LIN {X 0,Y 446.497,Z 325.867,A -85,B 0,C 180,E1 -8839.301,E2 -8839.301} C_VEL
LIN {X 0,Y 446.419,Z 325.877,A -85,B 0,C 180,E1 -8842.199,E2 -8842.199} C_VEL
LIN {X 0,Y 446.45,Z 325.872,A -85,B 0,C 180,E1 -8845.152,E2 -8845.152} C_VEL
LIN {X 0,Y 446.485,Z 325.867,A -85,B 0,C 180,E1 -8848.178,E2 -8848.178} C_VEL
LIN {X 0,Y 446.418,Z 325.875,A -85,B 0,C 180,E1 -8851.774,E2 -8851.774} C_VEL
LIN {X 0,Y 446.422,Z 325.878,A -85,B 0,C 180,E1 -8854.523,E2 -8854.523} C_VEL
LIN {X 0,Y 446.412,Z 325.876,A -85,B 0,C 180,E1 -8858.078,E2 -8858.078} C_VEL
LIN {X 0,Y 446.425,Z 325.876,A -85,B 0,C 180,E1 -8860.917,E2 -8860.917} C_VEL
LIN {X 0,Y 446.398,Z 325.878,A -85,B 0,C 180,E1 -8863.846,E2 -8863.846} C_VEL
LIN {X 0,Y 446.397,Z 325.882,A -85,B 0,C 180,E1 -8866.403,E2 -8866.403} C_VEL
LIN {X 0,Y 446.425,Z 325.874,A -85,B 0,C 180,E1 -8869.082,E2 -8869.082} C_VEL
LIN {X 0,Y 446.429,Z 325.874,A -85,B 0,C 180,E1 -8871.918,E2 -8871.918} C_VEL
LIN {X 0,Y 446.428,Z 325.873,A -85,B 0,C 180,E1 -8875.477,E2 -8875.477} C_VEL
LIN {X 0,Y 446.414,Z 325.878,A -85,B 0,C 180,E1 -8878.699,E2 -8878.699} C_VEL
LIN {X 0,Y 446.482,Z 325.868,A -85,B 0,C 180,E1 -8881.821,E2 -8881.821} C_VEL
LIN {X 0,Y 446.455,Z 325.871,A -85,B 0,C 180,E1 -8884.848,E2 -8884.848} C_VEL
LIN {X 0,Y 446.445,Z 325.876,A -85,B 0,C 180,E1 -8888.245,E2 -8888.245} C_VEL
LIN {X 0,Y 446.455,Z 325.871,A -85,B 0,C 180,E1 -8891.649,E2 -8891.649} C_VEL
LIN {X 0,Y 446.505,Z 325.868,A -85,B 0,C 180,E1 -8894.48,E2 -8894.48} C_VEL
LIN {X 0,Y 446.466,Z 325.869,A -85,B 0,C 180,E1 -8895.187,E2 -8895.187} C_VEL
LIN {X 0,Y 445.802,Z 325.955,A -85,B 0,C 180,E1 -8895.94,E2 -8895.94} C_VEL
LIN {X 0,Y 442.952,Z 326.308,A -85,B 0,C 180,E1 -8897.164,E2 -8897.164} C_VEL
LIN {X 0,Y 440.542,Z 326.611,A -85,B 0,C 180,E1 -8898.152,E2 -8898.152} C_VEL
LIN {X 0,Y 439.512,Z 326.735,A -85,B 0,C 180,E1 -8898.915,E2 -8898.915} C_VEL
LIN {X 0,Y 439.43,Z 326.745,A -85,B 0,C 180,E1 -8899.173,E2 -8899.173} C_VEL
LIN {X 0,Y 439.599,Z 326.726,A -85,B 0,C 180,E1 -8902.652,E2 -8902.652} C_VEL
LIN {X 0,Y 439.618,Z 326.725,A -85,B 0,C 180,E1 -8904.496,E2 -8904.496} C_VEL
LIN {X 0,Y 439.633,Z 326.725,A -85,B 0,C 180,E1 -8908.168,E2 -8908.168} C_VEL
LIN {X 0,Y 439.762,Z 326.708,A -85,B 0,C 180,E1 -8910,E2 -8910} C_VEL
LIN {X 0,Y 439.653,Z 326.718,A -85,B 0,C 180,E1 -8912.749,E2 -8912.749} C_VEL
LIN {X 0,Y 439.616,Z 326.725,A -85,B 0,C 180,E1 -8916.425,E2 -8916.425} C_VEL
LIN {X 0,Y 439.497,Z 326.738,A -85,B 0,C 180,E1 -8919.202,E2 -8919.202} C_VEL
LIN {X 0,Y 439.463,Z 326.741,A -85,B 0,C 180,E1 -8922.938,E2 -8922.938} C_VEL
LIN {X 0,Y 439.445,Z 326.746,A -85,B 0,C 180,E1 -8926.349,E2 -8926.349} C_VEL
LIN {X 0,Y 439.401,Z 326.751,A -85,B 0,C 180,E1 -8929.627,E2 -8929.627} C_VEL
LIN {X 0,Y 439.364,Z 326.754,A -85,B 0,C 180,E1 -8932.576,E2 -8932.576} C_VEL
LIN {X 0,Y 439.404,Z 326.751,A -85,B 0,C 180,E1 -8935.585,E2 -8935.585} C_VEL
LIN {X 0,Y 439.416,Z 326.747,A -85,B 0,C 180,E1 -8938.674,E2 -8938.674} C_VEL
LIN {X 0,Y 439.369,Z 326.757,A -85,B 0,C 180,E1 -8942.031,E2 -8942.031} C_VEL
LIN {X 0,Y 439.395,Z 326.751,A -85,B 0,C 180,E1 -8945.341,E2 -8945.341} C_VEL
LIN {X 0,Y 439.39,Z 326.751,A -85,B 0,C 180,E1 -8948.595,E2 -8948.595} C_VEL
LIN {X 0,Y 439.388,Z 326.752,A -85,B 0,C 180,E1 -8951.257,E2 -8951.257} C_VEL
LIN {X 0,Y 439.4,Z 326.75,A -85,B 0,C 180,E1 -8954.73,E2 -8954.73} C_VEL
LIN {X 0,Y 439.396,Z 326.755,A -85,B 0,C 180,E1 -8957.796,E2 -8957.796} C_VEL
LIN {X 0,Y 439.395,Z 326.751,A -85,B 0,C 180,E1 -8960.225,E2 -8960.225} C_VEL
LIN {X 0,Y 439.374,Z 326.758,A -85,B 0,C 180,E1 -8963.713,E2 -8963.713} C_VEL
LIN {X 0,Y 439.373,Z 326.754,A -85,B 0,C 180,E1 -8967.055,E2 -8967.055} C_VEL
LIN {X 0,Y 439.384,Z 326.752,A -85,B 0,C 180,E1 -8970.275,E2 -8970.275} C_VEL
LIN {X 0,Y 439.431,Z 326.749,A -85,B 0,C 180,E1 -8973.397,E2 -8973.397} C_VEL
LIN {X 0,Y 439.443,Z 326.743,A -85,B 0,C 180,E1 -8974.537,E2 -8974.537} C_VEL
LIN {X 0,Y 443.588,Z 339.182,A -85,B 0,C 180,E1 -8974.94,E2 -8974.94} C_VEL
LIN {X 0,Y 442.677,Z 414.373,A -85,B 0,C 180,E1 -8976.337,E2 -8976.337} C_VEL
LIN {X 0,Y 442.558,Z 425.989,A -85,B 0,C 180,E1 -8976.705,E2 -8976.705} C_VEL
LIN {X 0,Y 442.258,Z 438.78,A -85,B 0,C 180,E1 -8977.289,E2 -8977.289} C_VEL
LIN {X 0,Y 441.891,Z 451.182,A -85,B 0,C 180,E1 -8978.053,E2 -8978.053} C_VEL
LIN {X 0,Y 441.469,Z 461.829,A -85,B 0,C 180,E1 -8978.889,E2 -8978.889} C_VEL
LIN {X 0,Y 441.016,Z 472.96,A -85,B 0,C 180,E1 -8979.992,E2 -8979.992} C_VEL
LIN {X 0,Y 440.528,Z 482.488,A -85,B 0,C 180,E1 -8981.152,E2 -8981.152} C_VEL
LIN {X 0,Y 440.14,Z 490.434,A -85,B 0,C 180,E1 -8982.339,E2 -8982.339} C_VEL
LIN {X 0,Y 439.742,Z 498.632,A -85,B 0,C 180,E1 -8983.864,E2 -8983.864} C_VEL
LIN {X 0,Y 439.467,Z 504.268,A -85,B 0,C 180,E1 -8985.175,E2 -8985.175} C_VEL
LIN {X 0,Y 439.241,Z 509.068,A -85,B 0,C 180,E1 -8986.585,E2 -8986.585} C_VEL
LIN {X 0,Y 439.14,Z 512.67,A -85,B 0,C 180,E1 -8987.992,E2 -8987.992} C_VEL
LIN {X 0,Y 438.993,Z 514.461,A -85,B 0,C 180,E1 -8988.924,E2 -8988.924} C_VEL
LIN {X 0,Y 438.964,Z 515.833,A -85,B 0,C 180,E1 -8989.857,E2 -8989.857} C_VEL
LIN {X 0,Y 438.965,Z 516.774,A -85,B 0,C 180,E1 -8990.788,E2 -8990.788} C_VEL
LIN {X 0,Y 438.98,Z 517.257,A -85,B 0,C 180,E1 -8991.716,E2 -8991.716} C_VEL
LIN {X 0,Y 439.074,Z 517.293,A -85,B 0,C 180,E1 -8992.935,E2 -8992.935} C_VEL
LIN {X 0,Y 439.118,Z 516.257,A -85,B 0,C 180,E1 -8994.49,E2 -8994.49} C_VEL
LIN {X 0,Y 439.143,Z 515.092,A -85,B 0,C 180,E1 -8995.411,E2 -8995.411} C_VEL
LIN {X 0,Y 439.278,Z 512.524,A -85,B 0,C 180,E1 -8996.79,E2 -8996.79} C_VEL
LIN {X 0,Y 439.584,Z 508.903,A -85,B 0,C 180,E1 -8998.168,E2 -8998.168} C_VEL
LIN {X 0,Y 439.885,Z 504.163,A -85,B 0,C 180,E1 -8999.543,E2 -8999.543} C_VEL
LIN {X 0,Y 440.318,Z 498.125,A -85,B 0,C 180,E1 -9000.915,E2 -9000.915} C_VEL
LIN {X 0,Y 440.757,Z 490.589,A -85,B 0,C 180,E1 -9002.285,E2 -9002.285} C_VEL
LIN {X 0,Y 441.354,Z 481.185,A -85,B 0,C 180,E1 -9003.652,E2 -9003.652} C_VEL
LIN {X 0,Y 441.879,Z 471.347,A -85,B 0,C 180,E1 -9004.79,E2 -9004.79} C_VEL
LIN {X 0,Y 442.315,Z 460.406,A -85,B 0,C 180,E1 -9005.814,E2 -9005.814} C_VEL
LIN {X 0,Y 442.823,Z 449.541,A -85,B 0,C 180,E1 -9006.608,E2 -9006.608} C_VEL
LIN {X 0,Y 443.165,Z 436.449,A -85,B 0,C 180,E1 -9007.346,E2 -9007.346} C_VEL
LIN {X 0,Y 443.35,Z 423.637,A -85,B 0,C 180,E1 -9007.859,E2 -9007.859} C_VEL
LIN {X 0,Y 443.436,Z 410.181,A -85,B 0,C 180,E1 -9008.201,E2 -9008.201} C_VEL
LIN {X 0,Y 444.635,Z 339.873,A -85,B 0,C 180,E1 -9009.574,E2 -9009.574} C_VEL
LIN {X 0,Y 439.557,Z 327.4,A -85,B 0,C 180,E1 -9010.117,E2 -9010.117} C_VEL
LIN {X 0,Y 439.434,Z 326.752,A -85,B 0,C 180,E1 -9010.162,E2 -9010.162} C_VEL
LIN {X 0,Y 439.469,Z 326.745,A -85,B 0,C 180,E1 -9012.938,E2 -9012.938} C_VEL
LIN {X 0,Y 439.448,Z 326.747,A -85,B 0,C 180,E1 -9016.347,E2 -9016.347} C_VEL
LIN {X 0,Y 439.373,Z 326.757,A -85,B 0,C 180,E1 -9019.628,E2 -9019.628} C_VEL
LIN {X 0,Y 439.356,Z 326.757,A -85,B 0,C 180,E1 -9022.576,E2 -9022.576} C_VEL
LIN {X 0,Y 439.357,Z 326.757,A -85,B 0,C 180,E1 -9025.588,E2 -9025.588} C_VEL
LIN {X 0,Y 439.385,Z 326.753,A -85,B 0,C 180,E1 -9028.676,E2 -9028.676} C_VEL
LIN {X 0,Y 439.367,Z 326.757,A -85,B 0,C 180,E1 -9032.029,E2 -9032.029} C_VEL
LIN {X 0,Y 439.39,Z 326.748,A -85,B 0,C 180,E1 -9035.339,E2 -9035.339} C_VEL
LIN {X 0,Y 439.358,Z 326.753,A -85,B 0,C 180,E1 -9038.598,E2 -9038.598} C_VEL
LIN {X 0,Y 439.352,Z 326.756,A -85,B 0,C 180,E1 -9042.21,E2 -9042.21} C_VEL
LIN {X 0,Y 439.38,Z 326.753,A -85,B 0,C 180,E1 -9045.267,E2 -9045.267} C_VEL
LIN {X 0,Y 439.371,Z 326.752,A -85,B 0,C 180,E1 -9048.746,E2 -9048.746} C_VEL
LIN {X 0,Y 439.367,Z 326.758,A -85,B 0,C 180,E1 -9051.61,E2 -9051.61} C_VEL
LIN {X 0,Y 439.399,Z 326.75,A -85,B 0,C 180,E1 -9054.844,E2 -9054.844} C_VEL
LIN {X 0,Y 439.376,Z 326.754,A -85,B 0,C 180,E1 -9058.139,E2 -9058.139} C_VEL
LIN {X 0,Y 439.421,Z 326.85,A -85,B 0,C 180,E1 -9059.249,E2 -9059.249} C_VEL
LIN {X 0,Y 443.204,Z 343.947,A -85,B 0,C 180,E1 -9062.109,E2 -9062.109} C_VEL
LIN {X 0,Y 443.563,Z 347.321,A -85,B 0,C 180,E1 -9062.646,E2 -9062.646} C_VEL
LIN {X 0,Y 442.316,Z 368.721,A -85,B 0,C 180,E1 -9065.849,E2 -9065.849} C_VEL
LIN {X 0,Y 441.289,Z 388.385,A -85,B 0,C 180,E1 -9068.757,E2 -9068.757} C_VEL
LIN {X 0,Y 440.388,Z 409.595,A -85,B 0,C 180,E1 -9071.869,E2 -9071.869} C_VEL
LIN {X 0,Y 440.361,Z 410.41,A -85,B 0,C 180,E1 -9071.988,E2 -9071.988} C_VEL
LIN {X 0,Y 443.42,Z 438.789,A -85,B 0,C 180,E1 -9072.667,E2 -9072.667} C_VEL
LIN {X 0,Y 442.262,Z 521.633,A -85,B 0,C 180,E1 -9074.238,E2 -9074.238} C_VEL
LIN {X 0,Y 441.733,Z 534.688,A -85,B 0,C 180,E1 -9074.662,E2 -9074.662} C_VEL
LIN {X 0,Y 441.242,Z 546.877,A -85,B 0,C 180,E1 -9075.235,E2 -9075.235} C_VEL
LIN {X 0,Y 440.562,Z 559.508,A -85,B 0,C 180,E1 -9076.038,E2 -9076.038} C_VEL
LIN {X 0,Y 439.985,Z 571.311,A -85,B 0,C 180,E1 -9077.001,E2 -9077.001} C_VEL
LIN {X 0,Y 439.692,Z 580.107,A -85,B 0,C 180,E1 -9077.89,E2 -9077.89} C_VEL
LIN {X 0,Y 439.273,Z 588.726,A -85,B 0,C 180,E1 -9078.931,E2 -9078.931} C_VEL
LIN {X 0,Y 438.883,Z 598.064,A -85,B 0,C 180,E1 -9080.32,E2 -9080.32} C_VEL
LIN {X 0,Y 438.701,Z 605.586,A -85,B 0,C 180,E1 -9081.71,E2 -9081.71} C_VEL
LIN {X 0,Y 438.643,Z 611.595,A -85,B 0,C 180,E1 -9083.099,E2 -9083.099} C_VEL
LIN {X 0,Y 438.6,Z 616.273,A -85,B 0,C 180,E1 -9084.483,E2 -9084.483} C_VEL
LIN {X 0,Y 438.706,Z 618.729,A -85,B 0,C 180,E1 -9085.406,E2 -9085.406} C_VEL
LIN {X 0,Y 438.79,Z 620.721,A -85,B 0,C 180,E1 -9086.327,E2 -9086.327} C_VEL
LIN {X 0,Y 438.681,Z 622.237,A -85,B 0,C 180,E1 -9087.245,E2 -9087.245} C_VEL
LIN {X 0,Y 438.655,Z 623.274,A -85,B 0,C 180,E1 -9088.164,E2 -9088.164} C_VEL
LIN {X 0,Y 438.669,Z 623.889,A -85,B 0,C 180,E1 -9089.082,E2 -9089.082} C_VEL
LIN {X 0,Y 438.698,Z 624.084,A -85,B 0,C 180,E1 -9090,E2 -9090} C_VEL
LIN {X 0,Y 438.675,Z 623.83,A -85,B 0,C 180,E1 -9090.918,E2 -9090.918} C_VEL
LIN {X 0,Y 438.67,Z 623.115,A -85,B 0,C 180,E1 -9091.836,E2 -9091.836} C_VEL
LIN {X 0,Y 438.699,Z 621.982,A -85,B 0,C 180,E1 -9092.755,E2 -9092.755} C_VEL
LIN {X 0,Y 438.747,Z 619.435,A -85,B 0,C 180,E1 -9094.133,E2 -9094.133} C_VEL
LIN {X 0,Y 438.653,Z 615.806,A -85,B 0,C 180,E1 -9095.516,E2 -9095.516} C_VEL
LIN {X 0,Y 438.676,Z 610.23,A -85,B 0,C 180,E1 -9097.109,E2 -9097.109} C_VEL
LIN {X 0,Y 438.775,Z 603.838,A -85,B 0,C 180,E1 -9098.52,E2 -9098.52} C_VEL
LIN {X 0,Y 438.915,Z 595.986,A -85,B 0,C 180,E1 -9099.912,E2 -9099.912} C_VEL
LIN {X 0,Y 439.305,Z 586.319,A -85,B 0,C 180,E1 -9101.302,E2 -9101.302} C_VEL
LIN {X 0,Y 439.832,Z 576.403,A -85,B 0,C 180,E1 -9102.45,E2 -9102.45} C_VEL
LIN {X 0,Y 440.242,Z 567.168,A -85,B 0,C 180,E1 -9103.337,E2 -9103.337} C_VEL
LIN {X 0,Y 440.754,Z 556.383,A -85,B 0,C 180,E1 -9104.191,E2 -9104.191} C_VEL
LIN {X 0,Y 441.517,Z 543.551,A -85,B 0,C 180,E1 -9104.991,E2 -9104.991} C_VEL
LIN {X 0,Y 442.098,Z 530.571,A -85,B 0,C 180,E1 -9105.59,E2 -9105.59} C_VEL
LIN {X 0,Y 442.691,Z 516.243,A -85,B 0,C 180,E1 -9106.042,E2 -9106.042} C_VEL
LIN {X 0,Y 443.861,Z 437.805,A -85,B 0,C 180,E1 -9107.594,E2 -9107.594} C_VEL
LIN {X 0,Y 441.293,Z 411.851,A -85,B 0,C 180,E1 -9108.282,E2 -9108.282} C_VEL
LIN {X 0,Y 440.287,Z 404.18,A -85,B 0,C 180,E1 -9108.518,E2 -9108.518} C_VEL
LIN {X 0,Y 441.456,Z 379.504,A -85,B 0,C 180,E1 -9112.216,E2 -9112.216} C_VEL
LIN {X 0,Y 442.689,Z 357.498,A -85,B 0,C 180,E1 -9115.633,E2 -9115.633} C_VEL
LIN {X 0,Y 443.47,Z 345.209,A -85,B 0,C 180,E1 -9117.616,E2 -9117.616} C_VEL
LIN {X 0,Y 441.409,Z 334.678,A -85,B 0,C 180,E1 -9119.576,E2 -9119.576} C_VEL
LIN {X 0,Y 439.406,Z 326.756,A -85,B 0,C 180,E1 -9121.186,E2 -9121.186} C_VEL
LIN {X 0,Y 439.387,Z 326.756,A -85,B 0,C 180,E1 -9124.044,E2 -9124.044} C_VEL
LIN {X 0,Y 439.349,Z 326.759,A -85,B 0,C 180,E1 -9126.886,E2 -9126.886} C_VEL
LIN {X 0,Y 439.35,Z 326.76,A -85,B 0,C 180,E1 -9129.84,E2 -9129.84} C_VEL
LIN {X 0,Y 439.345,Z 326.76,A -85,B 0,C 180,E1 -9132.621,E2 -9132.621} C_VEL
LIN {X 0,Y 439.4,Z 326.751,A -85,B 0,C 180,E1 -9135.27,E2 -9135.27} C_VEL
LIN {X 0,Y 439.358,Z 326.755,A -85,B 0,C 180,E1 -9139.016,E2 -9139.016} C_VEL
LIN {X 0,Y 439.337,Z 326.757,A -85,B 0,C 180,E1 -9142.563,E2 -9142.563} C_VEL
LIN {X 0,Y 439.393,Z 326.75,A -85,B 0,C 180,E1 -9144.843,E2 -9144.843} C_VEL
LIN {X 0,Y 439.368,Z 326.757,A -85,B 0,C 180,E1 -9148.139,E2 -9148.139} C_VEL
LIN {X 0,Y 439.388,Z 326.755,A -85,B 0,C 180,E1 -9151.609,E2 -9151.609} C_VEL
LIN {X 0,Y 439.355,Z 326.758,A -85,B 0,C 180,E1 -9154.412,E2 -9154.412} C_VEL
LIN {X 0,Y 439.355,Z 326.761,A -85,B 0,C 180,E1 -9157.424,E2 -9157.424} C_VEL
LIN {X 0,Y 439.388,Z 326.754,A -85,B 0,C 180,E1 -9160.684,E2 -9160.684} C_VEL
LIN {X 0,Y 439.473,Z 326.747,A -85,B 0,C 180,E1 -9163.835,E2 -9163.835} C_VEL
LIN {X 0,Y 440.548,Z 329.721,A -85,B 0,C 180,E1 -9163.975,E2 -9163.975} C_VEL
LIN {X 0,Y 444.907,Z 340.719,A -85,B 0,C 180,E1 -9164.47,E2 -9164.47} C_VEL
LIN {X 0,Y 443.421,Z 417.623,A -85,B 0,C 180,E1 -9166.042,E2 -9166.042} C_VEL
LIN {X 0,Y 443.277,Z 431.324,A -85,B 0,C 180,E1 -9166.505,E2 -9166.505} C_VEL
LIN {X 0,Y 443.021,Z 443.747,A -85,B 0,C 180,E1 -9167.109,E2 -9167.109} C_VEL
LIN {X 0,Y 442.706,Z 455.181,A -85,B 0,C 180,E1 -9167.857,E2 -9167.857} C_VEL
LIN {X 0,Y 442.146,Z 466.263,A -85,B 0,C 180,E1 -9168.771,E2 -9168.771} C_VEL
LIN {X 0,Y 441.664,Z 476.26,A -85,B 0,C 180,E1 -9169.803,E2 -9169.803} C_VEL
LIN {X 0,Y 441.182,Z 484.458,A -85,B 0,C 180,E1 -9170.833,E2 -9170.833} C_VEL
LIN {X 0,Y 440.621,Z 493.308,A -85,B 0,C 180,E1 -9172.208,E2 -9172.208} C_VEL
LIN {X 0,Y 440.208,Z 500.393,A -85,B 0,C 180,E1 -9173.583,E2 -9173.583} C_VEL
LIN {X 0,Y 439.806,Z 506.032,A -85,B 0,C 180,E1 -9174.957,E2 -9174.957} C_VEL
LIN {X 0,Y 439.444,Z 510.432,A -85,B 0,C 180,E1 -9176.332,E2 -9176.332} C_VEL
LIN {X 0,Y 439.271,Z 512.716,A -85,B 0,C 180,E1 -9177.248,E2 -9177.248} C_VEL
LIN {X 0,Y 439.295,Z 514.538,A -85,B 0,C 180,E1 -9178.166,E2 -9178.166} C_VEL
LIN {X 0,Y 439.151,Z 515.963,A -85,B 0,C 180,E1 -9179.083,E2 -9179.083} C_VEL
LIN {X 0,Y 439.083,Z 516.914,A -85,B 0,C 180,E1 -9180,E2 -9180} C_VEL
LIN {X 0,Y 439.069,Z 517.457,A -85,B 0,C 180,E1 -9180.917,E2 -9180.917} C_VEL
LIN {X 0,Y 438.841,Z 517.636,A -85,B 0,C 180,E1 -9181.835,E2 -9181.835} C_VEL
LIN {X 0,Y 438.868,Z 517.357,A -85,B 0,C 180,E1 -9182.753,E2 -9182.753} C_VEL
LIN {X 0,Y 439.079,Z 515.522,A -85,B 0,C 180,E1 -9184.59,E2 -9184.59} C_VEL
LIN {X 0,Y 439.171,Z 513.052,A -85,B 0,C 180,E1 -9185.97,E2 -9185.97} C_VEL
LIN {X 0,Y 439.307,Z 509.56,A -85,B 0,C 180,E1 -9187.353,E2 -9187.353} C_VEL
LIN {X 0,Y 439.482,Z 504.951,A -85,B 0,C 180,E1 -9188.738,E2 -9188.738} C_VEL
LIN {X 0,Y 439.724,Z 499.09,A -85,B 0,C 180,E1 -9190.125,E2 -9190.125} C_VEL
LIN {X 0,Y 440.091,Z 491.706,A -85,B 0,C 180,E1 -9191.514,E2 -9191.514} C_VEL
LIN {X 0,Y 440.535,Z 482.494,A -85,B 0,C 180,E1 -9192.905,E2 -9192.905} C_VEL
LIN {X 0,Y 440.919,Z 472.98,A -85,B 0,C 180,E1 -9194.068,E2 -9194.068} C_VEL
LIN {X 0,Y 441.452,Z 462.355,A -85,B 0,C 180,E1 -9195.111,E2 -9195.111} C_VEL
LIN {X 0,Y 441.831,Z 450.551,A -85,B 0,C 180,E1 -9196.044,E2 -9196.044} C_VEL
LIN {X 0,Y 442.304,Z 438.038,A -85,B 0,C 180,E1 -9196.797,E2 -9196.797} C_VEL
LIN {X 0,Y 442.521,Z 424.952,A -85,B 0,C 180,E1 -9197.384,E2 -9197.384} C_VEL
LIN {X 0,Y 442.633,Z 412.315,A -85,B 0,C 180,E1 -9197.766,E2 -9197.766} C_VEL
LIN {X 0,Y 443.576,Z 339.103,A -85,B 0,C 180,E1 -9199.137,E2 -9199.137} C_VEL
LIN {X 0,Y 439.436,Z 326.746,A -85,B 0,C 180,E1 -9199.535,E2 -9199.535} C_VEL
LIN {X 0,Y 439.366,Z 326.758,A -85,B 0,C 180,E1 -9202.575,E2 -9202.575} C_VEL
LIN {X 0,Y 439.401,Z 326.748,A -85,B 0,C 180,E1 -9205.585,E2 -9205.585} C_VEL
LIN {X 0,Y 439.417,Z 326.752,A -85,B 0,C 180,E1 -9208.673,E2 -9208.673} C_VEL
LIN {X 0,Y 439.368,Z 326.753,A -85,B 0,C 180,E1 -9212.03,E2 -9212.03} C_VEL
LIN {X 0,Y 439.391,Z 326.75,A -85,B 0,C 180,E1 -9215.339,E2 -9215.339} C_VEL
LIN {X 0,Y 439.374,Z 326.758,A -85,B 0,C 180,E1 -9218.595,E2 -9218.595} C_VEL
LIN {X 0,Y 439.387,Z 326.751,A -85,B 0,C 180,E1 -9221.256,E2 -9221.256} C_VEL
LIN {X 0,Y 439.398,Z 326.753,A -85,B 0,C 180,E1 -9224.729,E2 -9224.729} C_VEL
LIN {X 0,Y 439.394,Z 326.75,A -85,B 0,C 180,E1 -9227.795,E2 -9227.795} C_VEL
LIN {X 0,Y 439.435,Z 326.747,A -85,B 0,C 180,E1 -9230.228,E2 -9230.228} C_VEL
LIN {X 0,Y 439.375,Z 326.752,A -85,B 0,C 180,E1 -9233.713,E2 -9233.713} C_VEL
LIN {X 0,Y 439.37,Z 326.753,A -85,B 0,C 180,E1 -9237.054,E2 -9237.054} C_VEL
LIN {X 0,Y 439.38,Z 326.755,A -85,B 0,C 180,E1 -9240.274,E2 -9240.274} C_VEL
LIN {X 0,Y 439.427,Z 326.746,A -85,B 0,C 180,E1 -9243.396,E2 -9243.396} C_VEL
LIN {X 0,Y 439.385,Z 326.756,A -85,B 0,C 180,E1 -9246.43,E2 -9246.43} C_VEL
LIN {X 0,Y 439.386,Z 326.751,A -85,B 0,C 180,E1 -9249.397,E2 -9249.397} C_VEL
LIN {X 0,Y 439.429,Z 326.751,A -85,B 0,C 180,E1 -9252.309,E2 -9252.309} C_VEL
LIN {X 0,Y 439.445,Z 326.743,A -85,B 0,C 180,E1 -9255.176,E2 -9255.176} C_VEL
LIN {X 0,Y 439.481,Z 326.742,A -85,B 0,C 180,E1 -9258.001,E2 -9258.001} C_VEL
LIN {X 0,Y 439.43,Z 326.745,A -85,B 0,C 180,E1 -9259.173,E2 -9259.173} C_VEL
LIN {X 0,Y 438.78,Z 326.83,A -85,B 0,C 180,E1 -9259.939,E2 -9259.939} C_VEL
LIN {X 0,Y 435.978,Z 327.175,A -85,B 0,C 180,E1 -9261.184,E2 -9261.184} C_VEL
LIN {X 0,Y 433.619,Z 327.474,A -85,B 0,C 180,E1 -9262.189,E2 -9262.189} C_VEL
LIN {X 0,Y 432.627,Z 327.593,A -85,B 0,C 180,E1 -9262.965,E2 -9262.965} C_VEL
LIN {X 0,Y 432.557,Z 327.601,A -85,B 0,C 180,E1 -9263.227,E2 -9263.227} C_VEL
LIN {X 0,Y 432.398,Z 327.622,A -85,B 0,C 180,E1 -9265.339,E2 -9265.339} C_VEL
LIN {X 0,Y 432.603,Z 327.6,A -85,B 0,C 180,E1 -9268.138,E2 -9268.138} C_VEL
LIN {X 0,Y 432.731,Z 327.583,A -85,B 0,C 180,E1 -9270,E2 -9270} C_VEL
LIN {X 0,Y 432.602,Z 327.596,A -85,B 0,C 180,E1 -9272.794,E2 -9272.794} C_VEL
LIN {X 0,Y 432.57,Z 327.602,A -85,B 0,C 180,E1 -9276.531,E2 -9276.531} C_VEL
LIN {X 0,Y 432.44,Z 327.617,A -85,B 0,C 180,E1 -9279.353,E2 -9279.353} C_VEL
LIN {X 0,Y 432.428,Z 327.618,A -85,B 0,C 180,E1 -9282.804,E2 -9282.804} C_VEL
LIN {X 0,Y 432.41,Z 327.621,A -85,B 0,C 180,E1 -9286.479,E2 -9286.479} C_VEL
LIN {X 0,Y 432.337,Z 327.634,A -85,B 0,C 180,E1 -9289.961,E2 -9289.961} C_VEL
LIN {X 0,Y 432.318,Z 327.632,A -85,B 0,C 180,E1 -9292.965,E2 -9292.965} C_VEL
LIN {X 0,Y 432.363,Z 327.63,A -85,B 0,C 180,E1 -9296.033,E2 -9296.033} C_VEL
LIN {X 0,Y 432.342,Z 327.629,A -85,B 0,C 180,E1 -9299.188,E2 -9299.188} C_VEL
LIN {X 0,Y 432.322,Z 327.632,A -85,B 0,C 180,E1 -9302.443,E2 -9302.443} C_VEL
LIN {X 0,Y 432.345,Z 327.631,A -85,B 0,C 180,E1 -9305.633,E2 -9305.633} C_VEL
LIN {X 0,Y 432.352,Z 327.628,A -85,B 0,C 180,E1 -9308.717,E2 -9308.717} C_VEL
LIN {X 0,Y 432.334,Z 327.634,A -85,B 0,C 180,E1 -9311.798,E2 -9311.798} C_VEL
LIN {X 0,Y 432.333,Z 327.63,A -85,B 0,C 180,E1 -9314.348,E2 -9314.348} C_VEL
LIN {X 0,Y 432.32,Z 327.632,A -85,B 0,C 180,E1 -9317.016,E2 -9317.016} C_VEL
LIN {X 0,Y 432.334,Z 327.634,A -85,B 0,C 180,E1 -9319.821,E2 -9319.821} C_VEL
LIN {X 0,Y 432.307,Z 327.634,A -85,B 0,C 180,E1 -9323.023,E2 -9323.023} C_VEL
LIN {X 0,Y 432.359,Z 327.629,A -85,B 0,C 180,E1 -9325.998,E2 -9325.998} C_VEL
LIN {X 0,Y 432.349,Z 327.631,A -85,B 0,C 180,E1 -9329.49,E2 -9329.49} C_VEL
LIN {X 0,Y 432.393,Z 327.624,A -85,B 0,C 180,E1 -9332.929,E2 -9332.929} C_VEL
LIN {X 0,Y 432.45,Z 327.759,A -85,B 0,C 180,E1 -9334.315,E2 -9334.315} C_VEL
LIN {X 0,Y 436.747,Z 340.599,A -85,B 0,C 180,E1 -9334.725,E2 -9334.725} C_VEL
LIN {X 0,Y 435.769,Z 414.594,A -85,B 0,C 180,E1 -9336.128,E2 -9336.128} C_VEL
LIN {X 0,Y 435.651,Z 425.89,A -85,B 0,C 180,E1 -9336.484,E2 -9336.484} C_VEL
LIN {X 0,Y 435.375,Z 438.76,A -85,B 0,C 180,E1 -9337.066,E2 -9337.066} C_VEL
LIN {X 0,Y 434.987,Z 450.886,A -85,B 0,C 180,E1 -9337.811,E2 -9337.811} C_VEL
LIN {X 0,Y 434.548,Z 461.754,A -85,B 0,C 180,E1 -9338.661,E2 -9338.661} C_VEL
LIN {X 0,Y 434.129,Z 471.956,A -85,B 0,C 180,E1 -9339.654,E2 -9339.654} C_VEL
LIN {X 0,Y 433.612,Z 481.837,A -85,B 0,C 180,E1 -9340.84,E2 -9340.84} C_VEL
LIN {X 0,Y 433.179,Z 490.076,A -85,B 0,C 180,E1 -9342.046,E2 -9342.046} C_VEL
LIN {X 0,Y 432.817,Z 497.339,A -85,B 0,C 180,E1 -9343.343,E2 -9343.343} C_VEL
LIN {X 0,Y 432.465,Z 504.372,A -85,B 0,C 180,E1 -9344.929,E2 -9344.929} C_VEL
LIN {X 0,Y 432.224,Z 509.346,A -85,B 0,C 180,E1 -9346.363,E2 -9346.363} C_VEL
LIN {X 0,Y 432.108,Z 513.118,A -85,B 0,C 180,E1 -9347.794,E2 -9347.794} C_VEL
LIN {X 0,Y 431.981,Z 515.026,A -85,B 0,C 180,E1 -9348.742,E2 -9348.742} C_VEL
LIN {X 0,Y 431.934,Z 516.466,A -85,B 0,C 180,E1 -9349.69,E2 -9349.69} C_VEL
LIN {X 0,Y 431.937,Z 517.499,A -85,B 0,C 180,E1 -9350.636,E2 -9350.636} C_VEL
LIN {X 0,Y 431.954,Z 518.081,A -85,B 0,C 180,E1 -9351.58,E2 -9351.58} C_VEL
LIN {X 0,Y 432.039,Z 518.206,A -85,B 0,C 180,E1 -9352.884,E2 -9352.884} C_VEL
LIN {X 0,Y 432.08,Z 517.322,A -85,B 0,C 180,E1 -9354.4,E2 -9354.4} C_VEL
LIN {X 0,Y 432.111,Z 516.213,A -85,B 0,C 180,E1 -9355.336,E2 -9355.336} C_VEL
LIN {X 0,Y 432.184,Z 514.704,A -85,B 0,C 180,E1 -9356.271,E2 -9356.271} C_VEL
LIN {X 0,Y 432.485,Z 511.568,A -85,B 0,C 180,E1 -9357.672,E2 -9357.672} C_VEL
LIN {X 0,Y 432.771,Z 507.367,A -85,B 0,C 180,E1 -9359.07,E2 -9359.07} C_VEL
LIN {X 0,Y 433.241,Z 500.887,A -85,B 0,C 180,E1 -9360.698,E2 -9360.698} C_VEL
LIN {X 0,Y 433.696,Z 493.831,A -85,B 0,C 180,E1 -9362.09,E2 -9362.09} C_VEL
LIN {X 0,Y 434.24,Z 486.592,A -85,B 0,C 180,E1 -9363.248,E2 -9363.248} C_VEL
LIN {X 0,Y 434.79,Z 476.815,A -85,B 0,C 180,E1 -9364.52,E2 -9364.52} C_VEL
LIN {X 0,Y 435.351,Z 466.895,A -85,B 0,C 180,E1 -9365.559,E2 -9365.559} C_VEL
LIN {X 0,Y 435.832,Z 455.946,A -85,B 0,C 180,E1 -9366.482,E2 -9366.482} C_VEL
LIN {X 0,Y 436.345,Z 443.541,A -85,B 0,C 180,E1 -9367.287,E2 -9367.287} C_VEL
LIN {X 0,Y 436.512,Z 431.961,A -85,B 0,C 180,E1 -9367.866,E2 -9367.866} C_VEL
LIN {X 0,Y 436.704,Z 419.347,A -85,B 0,C 180,E1 -9368.299,E2 -9368.299} C_VEL
LIN {X 0,Y 437.072,Z 390.634,A -85,B 0,C 180,E1 -9368.892,E2 -9368.892} C_VEL
LIN {X 0,Y 438.047,Z 341.723,A -85,B 0,C 180,E1 -9369.885,E2 -9369.885} C_VEL
LIN {X 0,Y 432.417,Z 327.825,A -85,B 0,C 180,E1 -9370.517,E2 -9370.517} C_VEL
LIN {X 0,Y 432.402,Z 327.623,A -85,B 0,C 180,E1 -9373.153,E2 -9373.153} C_VEL
LIN {X 0,Y 432.398,Z 327.625,A -85,B 0,C 180,E1 -9376.47,E2 -9376.47} C_VEL
LIN {X 0,Y 432.307,Z 327.64,A -85,B 0,C 180,E1 -9379.962,E2 -9379.962} C_VEL
LIN {X 0,Y 432.305,Z 327.634,A -85,B 0,C 180,E1 -9382.965,E2 -9382.965} C_VEL
LIN {X 0,Y 432.31,Z 327.638,A -85,B 0,C 180,E1 -9386.036,E2 -9386.036} C_VEL
LIN {X 0,Y 432.325,Z 327.63,A -85,B 0,C 180,E1 -9389.189,E2 -9389.189} C_VEL
LIN {X 0,Y 432.324,Z 327.633,A -85,B 0,C 180,E1 -9392.443,E2 -9392.443} C_VEL
LIN {X 0,Y 432.336,Z 327.631,A -85,B 0,C 180,E1 -9395.818,E2 -9395.818} C_VEL
LIN {X 0,Y 432.303,Z 327.632,A -85,B 0,C 180,E1 -9399.348,E2 -9399.348} C_VEL
LIN {X 0,Y 432.307,Z 327.634,A -85,B 0,C 180,E1 -9401.801,E2 -9401.801} C_VEL
LIN {X 0,Y 432.335,Z 327.631,A -85,B 0,C 180,E1 -9404.348,E2 -9404.348} C_VEL
LIN {X 0,Y 432.311,Z 327.633,A -85,B 0,C 180,E1 -9407.018,E2 -9407.018} C_VEL
LIN {X 0,Y 432.294,Z 327.639,A -85,B 0,C 180,E1 -9409.828,E2 -9409.828} C_VEL
LIN {X 0,Y 432.307,Z 327.634,A -85,B 0,C 180,E1 -9413.022,E2 -9413.022} C_VEL
LIN {X 0,Y 432.361,Z 327.63,A -85,B 0,C 180,E1 -9415.997,E2 -9415.997} C_VEL
LIN {X 0,Y 432.393,Z 327.686,A -85,B 0,C 180,E1 -9419.004,E2 -9419.004} C_VEL
LIN {X 0,Y 436.1,Z 344.563,A -85,B 0,C 180,E1 -9421.876,E2 -9421.876} C_VEL
LIN {X 0,Y 436.642,Z 348.06,A -85,B 0,C 180,E1 -9422.448,E2 -9422.448} C_VEL
LIN {X 0,Y 435.345,Z 369.378,A -85,B 0,C 180,E1 -9425.691,E2 -9425.691} C_VEL
LIN {X 0,Y 434.296,Z 389.023,A -85,B 0,C 180,E1 -9428.647,E2 -9428.647} C_VEL
LIN {X 0,Y 433.405,Z 409.079,A -85,B 0,C 180,E1 -9431.612,E2 -9431.612} C_VEL
LIN {X 0,Y 436.552,Z 440.109,A -85,B 0,C 180,E1 -9432.438,E2 -9432.438} C_VEL
LIN {X 0,Y 435.333,Z 520.878,A -85,B 0,C 180,E1 -9434.041,E2 -9434.041} C_VEL
LIN {X 0,Y 434.807,Z 533.85,A -85,B 0,C 180,E1 -9434.472,E2 -9434.472} C_VEL
LIN {X 0,Y 434.296,Z 546.038,A -85,B 0,C 180,E1 -9435.054,E2 -9435.054} C_VEL
LIN {X 0,Y 433.601,Z 557.874,A -85,B 0,C 180,E1 -9435.809,E2 -9435.809} C_VEL
LIN {X 0,Y 433.063,Z 569.383,A -85,B 0,C 180,E1 -9436.748,E2 -9436.748} C_VEL
LIN {X 0,Y 432.638,Z 579.82,A -85,B 0,C 180,E1 -9437.808,E2 -9437.808} C_VEL
LIN {X 0,Y 432.152,Z 589.179,A -85,B 0,C 180,E1 -9438.984,E2 -9438.984} C_VEL
LIN {X 0,Y 431.784,Z 598.307,A -85,B 0,C 180,E1 -9440.396,E2 -9440.396} C_VEL
LIN {X 0,Y 431.626,Z 605.625,A -85,B 0,C 180,E1 -9441.809,E2 -9441.809} C_VEL
LIN {X 0,Y 431.564,Z 612.258,A -85,B 0,C 180,E1 -9443.454,E2 -9443.454} C_VEL
LIN {X 0,Y 431.552,Z 616.583,A -85,B 0,C 180,E1 -9444.861,E2 -9444.861} C_VEL
LIN {X 0,Y 431.745,Z 619.788,A -85,B 0,C 180,E1 -9446.267,E2 -9446.267} C_VEL
LIN {X 0,Y 431.634,Z 621.322,A -85,B 0,C 180,E1 -9447.2,E2 -9447.2} C_VEL
LIN {X 0,Y 431.606,Z 622.378,A -85,B 0,C 180,E1 -9448.134,E2 -9448.134} C_VEL
LIN {X 0,Y 431.621,Z 623.001,A -85,B 0,C 180,E1 -9449.067,E2 -9449.067} C_VEL
LIN {X 0,Y 431.653,Z 623.203,A -85,B 0,C 180,E1 -9450,E2 -9450} C_VEL
LIN {X 0,Y 431.625,Z 622.962,A -85,B 0,C 180,E1 -9450.933,E2 -9450.933} C_VEL
LIN {X 0,Y 431.617,Z 622.252,A -85,B 0,C 180,E1 -9451.866,E2 -9451.866} C_VEL
LIN {X 0,Y 431.649,Z 621.121,A -85,B 0,C 180,E1 -9452.8,E2 -9452.8} C_VEL
LIN {X 0,Y 431.68,Z 618.576,A -85,B 0,C 180,E1 -9454.201,E2 -9454.201} C_VEL
LIN {X 0,Y 431.594,Z 614.943,A -85,B 0,C 180,E1 -9455.607,E2 -9455.607} C_VEL
LIN {X 0,Y 431.596,Z 609.366,A -85,B 0,C 180,E1 -9457.226,E2 -9457.226} C_VEL
LIN {X 0,Y 431.688,Z 602.986,A -85,B 0,C 180,E1 -9458.661,E2 -9458.661} C_VEL
LIN {X 0,Y 431.851,Z 595.141,A -85,B 0,C 180,E1 -9460.075,E2 -9460.075} C_VEL
LIN {X 0,Y 432.244,Z 585.479,A -85,B 0,C 180,E1 -9461.489,E2 -9461.489} C_VEL
LIN {X 0,Y 432.84,Z 574.747,A -85,B 0,C 180,E1 -9462.745,E2 -9462.745} C_VEL
LIN {X 0,Y 433.403,Z 563.194,A -85,B 0,C 180,E1 -9463.838,E2 -9463.838} C_VEL
LIN {X 0,Y 434.053,Z 552.428,A -85,B 0,C 180,E1 -9464.655,E2 -9464.655} C_VEL
LIN {X 0,Y 434.828,Z 539.692,A -85,B 0,C 180,E1 -9465.407,E2 -9465.407} C_VEL
LIN {X 0,Y 435.491,Z 526.6,A -85,B 0,C 180,E1 -9465.983,E2 -9465.983} C_VEL
LIN {X 0,Y 435.952,Z 512.87,A -85,B 0,C 180,E1 -9466.387,E2 -9466.387} C_VEL
LIN {X 0,Y 437.222,Z 438.772,A -85,B 0,C 180,E1 -9467.892,E2 -9467.892} C_VEL
LIN {X 0,Y 434.701,Z 412.877,A -85,B 0,C 180,E1 -9468.604,E2 -9468.604} C_VEL
LIN {X 0,Y 433.36,Z 402.909,A -85,B 0,C 180,E1 -9468.926,E2 -9468.926} C_VEL
LIN {X 0,Y 434.592,Z 378.435,A -85,B 0,C 180,E1 -9472.681,E2 -9472.681} C_VEL
LIN {X 0,Y 435.854,Z 358.787,A -85,B 0,C 180,E1 -9475.809,E2 -9475.809} C_VEL
LIN {X 0,Y 436.653,Z 346.605,A -85,B 0,C 180,E1 -9477.824,E2 -9477.824} C_VEL
LIN {X 0,Y 434.241,Z 334.791,A -85,B 0,C 180,E1 -9480.114,E2 -9480.114} C_VEL
LIN {X 0,Y 432.338,Z 327.637,A -85,B 0,C 180,E1 -9481.686,E2 -9481.686} C_VEL
LIN {X 0,Y 432.339,Z 327.632,A -85,B 0,C 180,E1 -9484.677,E2 -9484.677} C_VEL
LIN {X 0,Y 432.332,Z 327.634,A -85,B 0,C 180,E1 -9488.151,E2 -9488.151} C_VEL
LIN {X 0,Y 432.311,Z 327.637,A -85,B 0,C 180,E1 -9491.8,E2 -9491.8} C_VEL
LIN {X 0,Y 432.336,Z 327.634,A -85,B 0,C 180,E1 -9494.347,E2 -9494.347} C_VEL
LIN {X 0,Y 432.309,Z 327.633,A -85,B 0,C 180,E1 -9497.018,E2 -9497.018} C_VEL
LIN {X 0,Y 432.291,Z 327.638,A -85,B 0,C 180,E1 -9499.828,E2 -9499.828} C_VEL
LIN {X 0,Y 432.298,Z 327.633,A -85,B 0,C 180,E1 -9503.021,E2 -9503.021} C_VEL
LIN {X 0,Y 432.334,Z 327.633,A -85,B 0,C 180,E1 -9506.002,E2 -9506.002} C_VEL
LIN {X 0,Y 432.343,Z 327.632,A -85,B 0,C 180,E1 -9509.491,E2 -9509.491} C_VEL
LIN {X 0,Y 432.319,Z 327.636,A -85,B 0,C 180,E1 -9511.872,E2 -9511.872} C_VEL
LIN {X 0,Y 432.347,Z 327.634,A -85,B 0,C 180,E1 -9515.548,E2 -9515.548} C_VEL
LIN {X 0,Y 432.336,Z 327.634,A -85,B 0,C 180,E1 -9519.045,E2 -9519.045} C_VEL
LIN {X 0,Y 432.341,Z 327.633,A -85,B 0,C 180,E1 -9522.009,E2 -9522.009} C_VEL
LIN {X 0,Y 432.414,Z 327.808,A -85,B 0,C 180,E1 -9523.432,E2 -9523.432} C_VEL
LIN {X 0,Y 433.517,Z 330.664,A -85,B 0,C 180,E1 -9523.572,E2 -9523.572} C_VEL
LIN {X 0,Y 438.329,Z 342.103,A -85,B 0,C 180,E1 -9524.133,E2 -9524.133} C_VEL
LIN {X 0,Y 436.739,Z 418.039,A -85,B 0,C 180,E1 -9525.734,E2 -9525.734} C_VEL
LIN {X 0,Y 436.639,Z 431.23,A -85,B 0,C 180,E1 -9526.177,E2 -9526.177} C_VEL
LIN {X 0,Y 436.338,Z 443.879,A -85,B 0,C 180,E1 -9526.79,E2 -9526.79} C_VEL
LIN {X 0,Y 436.008,Z 455.533,A -85,B 0,C 180,E1 -9527.549,E2 -9527.549} C_VEL
LIN {X 0,Y 435.401,Z 466.71,A -85,B 0,C 180,E1 -9528.477,E2 -9528.477} C_VEL
LIN {X 0,Y 434.903,Z 476.798,A -85,B 0,C 180,E1 -9529.525,E2 -9529.525} C_VEL
LIN {X 0,Y 434.33,Z 485.891,A -85,B 0,C 180,E1 -9530.687,E2 -9530.687} C_VEL
LIN {X 0,Y 433.705,Z 494.653,A -85,B 0,C 180,E1 -9532.083,E2 -9532.083} C_VEL
LIN {X 0,Y 433.268,Z 501.66,A -85,B 0,C 180,E1 -9533.48,E2 -9533.48} C_VEL
LIN {X 0,Y 432.829,Z 507.23,A -85,B 0,C 180,E1 -9534.876,E2 -9534.876} C_VEL
LIN {X 0,Y 432.47,Z 511.555,A -85,B 0,C 180,E1 -9536.273,E2 -9536.273} C_VEL
LIN {X 0,Y 432.275,Z 513.806,A -85,B 0,C 180,E1 -9537.204,E2 -9537.204} C_VEL
LIN {X 0,Y 432.291,Z 515.595,A -85,B 0,C 180,E1 -9538.136,E2 -9538.136} C_VEL
LIN {X 0,Y 432.149,Z 516.969,A -85,B 0,C 180,E1 -9539.068,E2 -9539.068} C_VEL
LIN {X 0,Y 432.055,Z 517.883,A -85,B 0,C 180,E1 -9540,E2 -9540} C_VEL
LIN {X 0,Y 432.037,Z 518.394,A -85,B 0,C 180,E1 -9540.932,E2 -9540.932} C_VEL
LIN {X 0,Y 431.8,Z 518.539,A -85,B 0,C 180,E1 -9541.865,E2 -9541.865} C_VEL
LIN {X 0,Y 431.823,Z 518.201,A -85,B 0,C 180,E1 -9542.798,E2 -9542.798} C_VEL
LIN {X 0,Y 431.899,Z 517.447,A -85,B 0,C 180,E1 -9543.732,E2 -9543.732} C_VEL
LIN {X 0,Y 432.056,Z 516.287,A -85,B 0,C 180,E1 -9544.665,E2 -9544.665} C_VEL
LIN {X 0,Y 432.152,Z 513.74,A -85,B 0,C 180,E1 -9546.068,E2 -9546.068} C_VEL
LIN {X 0,Y 432.284,Z 510.167,A -85,B 0,C 180,E1 -9547.473,E2 -9547.473} C_VEL
LIN {X 0,Y 432.469,Z 505.466,A -85,B 0,C 180,E1 -9548.881,E2 -9548.881} C_VEL
LIN {X 0,Y 432.742,Z 499.48,A -85,B 0,C 180,E1 -9550.29,E2 -9550.29} C_VEL
LIN {X 0,Y 433.108,Z 491.958,A -85,B 0,C 180,E1 -9551.702,E2 -9551.702} C_VEL
LIN {X 0,Y 433.58,Z 482.603,A -85,B 0,C 180,E1 -9553.116,E2 -9553.116} C_VEL
LIN {X 0,Y 433.993,Z 472.857,A -85,B 0,C 180,E1 -9554.297,E2 -9554.297} C_VEL
LIN {X 0,Y 434.511,Z 462.024,A -85,B 0,C 180,E1 -9555.358,E2 -9555.358} C_VEL
LIN {X 0,Y 434.869,Z 451.569,A -85,B 0,C 180,E1 -9556.187,E2 -9556.187} C_VEL
LIN {X 0,Y 435.341,Z 439.243,A -85,B 0,C 180,E1 -9556.948,E2 -9556.948} C_VEL
LIN {X 0,Y 435.611,Z 425.422,A -85,B 0,C 180,E1 -9557.578,E2 -9557.578} C_VEL
LIN {X 0,Y 435.705,Z 412.595,A -85,B 0,C 180,E1 -9557.967,E2 -9557.967} C_VEL
LIN {X 0,Y 436.599,Z 340.316,A -85,B 0,C 180,E1 -9559.36,E2 -9559.36} C_VEL
LIN {X 0,Y 432.387,Z 327.624,A -85,B 0,C 180,E1 -9559.777,E2 -9559.777} C_VEL
LIN {X 0,Y 432.32,Z 327.635,A -85,B 0,C 180,E1 -9562.964,E2 -9562.964} C_VEL
LIN {X 0,Y 432.363,Z 327.626,A -85,B 0,C 180,E1 -9566.032,E2 -9566.032} C_VEL
LIN {X 0,Y 432.343,Z 327.629,A -85,B 0,C 180,E1 -9569.187,E2 -9569.187} C_VEL
LIN {X 0,Y 432.322,Z 327.634,A -85,B 0,C 180,E1 -9572.442,E2 -9572.442} C_VEL
LIN {X 0,Y 432.342,Z 327.628,A -85,B 0,C 180,E1 -9575.631,E2 -9575.631} C_VEL
LIN {X 0,Y 432.337,Z 327.634,A -85,B 0,C 180,E1 -9578.714,E2 -9578.714} C_VEL
LIN {X 0,Y 432.332,Z 327.63,A -85,B 0,C 180,E1 -9581.797,E2 -9581.797} C_VEL
LIN {X 0,Y 432.332,Z 327.632,A -85,B 0,C 180,E1 -9584.347,E2 -9584.347} C_VEL
LIN {X 0,Y 432.318,Z 327.632,A -85,B 0,C 180,E1 -9587.015,E2 -9587.015} C_VEL
LIN {X 0,Y 432.339,Z 327.629,A -85,B 0,C 180,E1 -9589.819,E2 -9589.819} C_VEL
LIN {X 0,Y 432.313,Z 327.633,A -85,B 0,C 180,E1 -9593.023,E2 -9593.023} C_VEL
LIN {X 0,Y 432.357,Z 327.627,A -85,B 0,C 180,E1 -9595.996,E2 -9595.996} C_VEL
LIN {X 0,Y 432.345,Z 327.628,A -85,B 0,C 180,E1 -9599.489,E2 -9599.489} C_VEL
LIN {X 0,Y 432.39,Z 327.623,A -85,B 0,C 180,E1 -9602.928,E2 -9602.928} C_VEL
LIN {X 0,Y 432.369,Z 327.627,A -85,B 0,C 180,E1 -9606.023,E2 -9606.023} C_VEL
LIN {X 0,Y 432.347,Z 327.628,A -85,B 0,C 180,E1 -9609.046,E2 -9609.046} C_VEL
LIN {X 0,Y 432.375,Z 327.626,A -85,B 0,C 180,E1 -9612.011,E2 -9612.011} C_VEL
LIN {X 0,Y 432.393,Z 327.622,A -85,B 0,C 180,E1 -9614.926,E2 -9614.926} C_VEL
LIN {X 0,Y 432.456,Z 327.615,A -85,B 0,C 180,E1 -9617.803,E2 -9617.803} C_VEL
LIN {X 0,Y 432.489,Z 327.61,A -85,B 0,C 180,E1 -9621.59,E2 -9621.59} C_VEL
LIN {X 0,Y 432.557,Z 327.601,A -85,B 0,C 180,E1 -9623.227,E2 -9623.227} C_VEL
LIN {X 0,Y 431.922,Z 327.685,A -85,B 0,C 180,E1 -9624.002,E2 -9624.002} C_VEL
LIN {X 0,Y 429.091,Z 328.035,A -85,B 0,C 180,E1 -9625.262,E2 -9625.262} C_VEL
LIN {X 0,Y 426.676,Z 328.339,A -85,B 0,C 180,E1 -9626.279,E2 -9626.279} C_VEL
LIN {X 0,Y 425.635,Z 328.465,A -85,B 0,C 180,E1 -9627.065,E2 -9627.065} C_VEL
LIN {X 0,Y 425.549,Z 328.474,A -85,B 0,C 180,E1 -9627.331,E2 -9627.331} C_VEL
LIN {X 0,Y 425.701,Z 328.459,A -85,B 0,C 180,E1 -9630,E2 -9630} C_VEL
LIN {X 0,Y 425.554,Z 328.474,A -85,B 0,C 180,E1 -9632.84,E2 -9632.84} C_VEL
LIN {X 0,Y 425.529,Z 328.478,A -85,B 0,C 180,E1 -9636.639,E2 -9636.639} C_VEL
LIN {X 0,Y 425.399,Z 328.494,A -85,B 0,C 180,E1 -9639.51,E2 -9639.51} C_VEL
LIN {X 0,Y 425.391,Z 328.495,A -85,B 0,C 180,E1 -9642.904,E2 -9642.904} C_VEL
LIN {X 0,Y 425.359,Z 328.499,A -85,B 0,C 180,E1 -9646.605,E2 -9646.605} C_VEL
LIN {X 0,Y 425.327,Z 328.504,A -85,B 0,C 180,E1 -9649.636,E2 -9649.636} C_VEL
LIN {X 0,Y 425.306,Z 328.506,A -85,B 0,C 180,E1 -9653.366,E2 -9653.366} C_VEL
LIN {X 0,Y 425.347,Z 328.5,A -85,B 0,C 180,E1 -9656.845,E2 -9656.845} C_VEL
LIN {X 0,Y 425.29,Z 328.51,A -85,B 0,C 180,E1 -9659.72,E2 -9659.72} C_VEL
LIN {X 0,Y 425.281,Z 328.509,A -85,B 0,C 180,E1 -9663.049,E2 -9663.049} C_VEL
LIN {X 0,Y 425.284,Z 328.512,A -85,B 0,C 180,E1 -9665.93,E2 -9665.93} C_VEL
LIN {X 0,Y 425.303,Z 328.506,A -85,B 0,C 180,E1 -9669.045,E2 -9669.045} C_VEL
LIN {X 0,Y 425.274,Z 328.509,A -85,B 0,C 180,E1 -9672.654,E2 -9672.654} C_VEL
LIN {X 0,Y 425.261,Z 328.513,A -85,B 0,C 180,E1 -9676.045,E2 -9676.045} C_VEL
LIN {X 0,Y 425.274,Z 328.509,A -85,B 0,C 180,E1 -9678.622,E2 -9678.622} C_VEL
LIN {X 0,Y 425.298,Z 328.507,A -85,B 0,C 180,E1 -9681.102,E2 -9681.102} C_VEL
LIN {X 0,Y 425.299,Z 328.507,A -85,B 0,C 180,E1 -9684.665,E2 -9684.665} C_VEL
LIN {X 0,Y 425.265,Z 328.512,A -85,B 0,C 180,E1 -9688.074,E2 -9688.074} C_VEL
LIN {X 0,Y 425.333,Z 328.504,A -85,B 0,C 180,E1 -9691.369,E2 -9691.369} C_VEL
LIN {X 0,Y 425.375,Z 328.497,A -85,B 0,C 180,E1 -9694.056,E2 -9694.056} C_VEL
LIN {X 0,Y 429.882,Z 342.195,A -85,B 0,C 180,E1 -9694.506,E2 -9694.506} C_VEL
LIN {X 0,Y 428.852,Z 416.547,A -85,B 0,C 180,E1 -9695.956,E2 -9695.956} C_VEL
LIN {X 0,Y 428.755,Z 427.031,A -85,B 0,C 180,E1 -9696.303,E2 -9696.303} C_VEL
LIN {X 0,Y 428.476,Z 439.554,A -85,B 0,C 180,E1 -9696.882,E2 -9696.882} C_VEL
LIN {X 0,Y 428.041,Z 452.345,A -85,B 0,C 180,E1 -9697.686,E2 -9697.686} C_VEL
LIN {X 0,Y 427.583,Z 463.098,A -85,B 0,C 180,E1 -9698.549,E2 -9698.549} C_VEL
LIN {X 0,Y 427.154,Z 472.991,A -85,B 0,C 180,E1 -9699.536,E2 -9699.536} C_VEL
LIN {X 0,Y 426.598,Z 483.012,A -85,B 0,C 180,E1 -9700.763,E2 -9700.763} C_VEL
LIN {X 0,Y 426.183,Z 491.21,A -85,B 0,C 180,E1 -9701.99,E2 -9701.99} C_VEL
LIN {X 0,Y 425.793,Z 498.622,A -85,B 0,C 180,E1 -9703.352,E2 -9703.352} C_VEL
LIN {X 0,Y 425.472,Z 504.476,A -85,B 0,C 180,E1 -9704.676,E2 -9704.676} C_VEL
LIN {X 0,Y 425.214,Z 509.616,A -85,B 0,C 180,E1 -9706.134,E2 -9706.134} C_VEL
LIN {X 0,Y 425.083,Z 513.541,A -85,B 0,C 180,E1 -9707.589,E2 -9707.589} C_VEL
LIN {X 0,Y 424.973,Z 515.568,A -85,B 0,C 180,E1 -9708.554,E2 -9708.554} C_VEL
LIN {X 0,Y 424.889,Z 517.097,A -85,B 0,C 180,E1 -9709.517,E2 -9709.517} C_VEL
LIN {X 0,Y 424.883,Z 518.196,A -85,B 0,C 180,E1 -9710.479,E2 -9710.479} C_VEL
LIN {X 0,Y 424.913,Z 518.891,A -85,B 0,C 180,E1 -9711.44,E2 -9711.44} C_VEL
LIN {X 0,Y 425.012,Z 519.104,A -85,B 0,C 180,E1 -9712.825,E2 -9712.825} C_VEL
LIN {X 0,Y 425.043,Z 518.378,A -85,B 0,C 180,E1 -9714.307,E2 -9714.307} C_VEL
LIN {X 0,Y 425.081,Z 517.366,A -85,B 0,C 180,E1 -9715.259,E2 -9715.259} C_VEL
LIN {X 0,Y 425.156,Z 515.921,A -85,B 0,C 180,E1 -9716.209,E2 -9716.209} C_VEL
LIN {X 0,Y 425.466,Z 512.91,A -85,B 0,C 180,E1 -9717.634,E2 -9717.634} C_VEL
LIN {X 0,Y 425.778,Z 508.835,A -85,B 0,C 180,E1 -9719.055,E2 -9719.055} C_VEL
LIN {X 0,Y 426.184,Z 503.568,A -85,B 0,C 180,E1 -9720.473,E2 -9720.473} C_VEL
LIN {X 0,Y 426.668,Z 496.927,A -85,B 0,C 180,E1 -9721.888,E2 -9721.888} C_VEL
LIN {X 0,Y 427.31,Z 488.575,A -85,B 0,C 180,E1 -9723.3,E2 -9723.3} C_VEL
LIN {X 0,Y 427.859,Z 480.065,A -85,B 0,C 180,E1 -9724.475,E2 -9724.475} C_VEL
LIN {X 0,Y 428.437,Z 470.712,A -85,B 0,C 180,E1 -9725.531,E2 -9725.531} C_VEL
LIN {X 0,Y 428.91,Z 460.487,A -85,B 0,C 180,E1 -9726.469,E2 -9726.469} C_VEL
LIN {X 0,Y 429.46,Z 449.226,A -85,B 0,C 180,E1 -9727.287,E2 -9727.287} C_VEL
LIN {X 0,Y 429.787,Z 436.613,A -85,B 0,C 180,E1 -9727.99,E2 -9727.99} C_VEL
LIN {X 0,Y 429.996,Z 423.152,A -85,B 0,C 180,E1 -9728.518,E2 -9728.518} C_VEL
LIN {X 0,Y 430.12,Z 406.957,A -85,B 0,C 180,E1 -9728.901,E2 -9728.901} C_VEL
LIN {X 0,Y 431.473,Z 343.357,A -85,B 0,C 180,E1 -9730.217,E2 -9730.217} C_VEL
LIN {X 0,Y 425.416,Z 328.972,A -85,B 0,C 180,E1 -9730.922,E2 -9730.922} C_VEL
LIN {X 0,Y 425.347,Z 328.507,A -85,B 0,C 180,E1 -9730.943,E2 -9730.943} C_VEL
LIN {X 0,Y 425.35,Z 328.501,A -85,B 0,C 180,E1 -9733.375,E2 -9733.375} C_VEL
LIN {X 0,Y 425.35,Z 328.503,A -85,B 0,C 180,E1 -9736.598,E2 -9736.598} C_VEL
LIN {X 0,Y 425.296,Z 328.511,A -85,B 0,C 180,E1 -9739.622,E2 -9739.622} C_VEL
LIN {X 0,Y 425.289,Z 328.512,A -85,B 0,C 180,E1 -9742.339,E2 -9742.339} C_VEL
LIN {X 0,Y 425.255,Z 328.514,A -85,B 0,C 180,E1 -9745.448,E2 -9745.448} C_VEL
LIN {X 0,Y 425.304,Z 328.506,A -85,B 0,C 180,E1 -9748.858,E2 -9748.858} C_VEL
LIN {X 0,Y 425.265,Z 328.513,A -85,B 0,C 180,E1 -9751.927,E2 -9751.927} C_VEL
LIN {X 0,Y 425.296,Z 328.503,A -85,B 0,C 180,E1 -9755.337,E2 -9755.337} C_VEL
LIN {X 0,Y 425.28,Z 328.505,A -85,B 0,C 180,E1 -9758.901,E2 -9758.901} C_VEL
LIN {X 0,Y 425.26,Z 328.509,A -85,B 0,C 180,E1 -9762.655,E2 -9762.655} C_VEL
LIN {X 0,Y 425.287,Z 328.508,A -85,B 0,C 180,E1 -9765.283,E2 -9765.283} C_VEL
LIN {X 0,Y 425.255,Z 328.511,A -85,B 0,C 180,E1 -9768.619,E2 -9768.619} C_VEL
LIN {X 0,Y 425.284,Z 328.51,A -85,B 0,C 180,E1 -9771.099,E2 -9771.099} C_VEL
LIN {X 0,Y 425.301,Z 328.506,A -85,B 0,C 180,E1 -9774.664,E2 -9774.664} C_VEL
LIN {X 0,Y 425.279,Z 328.511,A -85,B 0,C 180,E1 -9778.074,E2 -9778.074} C_VEL
LIN {X 0,Y 425.344,Z 328.643,A -85,B 0,C 180,E1 -9778.774,E2 -9778.774} C_VEL
LIN {X 0,Y 429.001,Z 345.16,A -85,B 0,C 180,E1 -9781.635,E2 -9781.635} C_VEL
LIN {X 0,Y 429.699,Z 349.475,A -85,B 0,C 180,E1 -9782.355,E2 -9782.355} C_VEL
LIN {X 0,Y 428.225,Z 373.274,A -85,B 0,C 180,E1 -9786.034,E2 -9786.034} C_VEL
LIN {X 0,Y 426.873,Z 398.645,A -85,B 0,C 180,E1 -9789.904,E2 -9789.904} C_VEL
LIN {X 0,Y 426.441,Z 407.093,A -85,B 0,C 180,E1 -9791.184,E2 -9791.184} C_VEL
LIN {X 0,Y 429.9,Z 439.951,A -85,B 0,C 180,E1 -9792.115,E2 -9792.115} C_VEL
LIN {X 0,Y 428.548,Z 516.346,A -85,B 0,C 180,E1 -9793.689,E2 -9793.689} C_VEL
LIN {X 0,Y 427.954,Z 530.731,A -85,B 0,C 180,E1 -9794.186,E2 -9794.186} C_VEL
LIN {X 0,Y 427.357,Z 544.019,A -85,B 0,C 180,E1 -9794.805,E2 -9794.805} C_VEL
LIN {X 0,Y 426.725,Z 556.212,A -85,B 0,C 180,E1 -9795.575,E2 -9795.575} C_VEL
LIN {X 0,Y 426.17,Z 566.551,A -85,B 0,C 180,E1 -9796.408,E2 -9796.408} C_VEL
LIN {X 0,Y 425.81,Z 575.13,A -85,B 0,C 180,E1 -9797.243,E2 -9797.243} C_VEL
LIN {X 0,Y 425.212,Z 584.314,A -85,B 0,C 180,E1 -9798.318,E2 -9798.318} C_VEL
LIN {X 0,Y 424.882,Z 592.758,A -85,B 0,C 180,E1 -9799.516,E2 -9799.516} C_VEL
LIN {X 0,Y 424.615,Z 601.025,A -85,B 0,C 180,E1 -9800.953,E2 -9800.953} C_VEL
LIN {X 0,Y 424.517,Z 607.626,A -85,B 0,C 180,E1 -9802.389,E2 -9802.389} C_VEL
LIN {X 0,Y 424.495,Z 612.497,A -85,B 0,C 180,E1 -9803.717,E2 -9803.717} C_VEL
LIN {X 0,Y 424.559,Z 616.803,A -85,B 0,C 180,E1 -9805.252,E2 -9805.252} C_VEL
LIN {X 0,Y 424.698,Z 618.836,A -85,B 0,C 180,E1 -9806.204,E2 -9806.204} C_VEL
LIN {X 0,Y 424.588,Z 620.387,A -85,B 0,C 180,E1 -9807.153,E2 -9807.153} C_VEL
LIN {X 0,Y 424.558,Z 621.473,A -85,B 0,C 180,E1 -9808.103,E2 -9808.103} C_VEL
LIN {X 0,Y 424.575,Z 622.106,A -85,B 0,C 180,E1 -9809.051,E2 -9809.051} C_VEL
LIN {X 0,Y 424.608,Z 622.317,A -85,B 0,C 180,E1 -9810,E2 -9810} C_VEL
LIN {X 0,Y 424.576,Z 622.09,A -85,B 0,C 180,E1 -9810.948,E2 -9810.948} C_VEL
LIN {X 0,Y 424.563,Z 621.389,A -85,B 0,C 180,E1 -9811.897,E2 -9811.897} C_VEL
LIN {X 0,Y 424.6,Z 620.262,A -85,B 0,C 180,E1 -9812.846,E2 -9812.846} C_VEL
LIN {X 0,Y 424.611,Z 617.725,A -85,B 0,C 180,E1 -9814.271,E2 -9814.271} C_VEL
LIN {X 0,Y 424.535,Z 614.103,A -85,B 0,C 180,E1 -9815.7,E2 -9815.7} C_VEL
LIN {X 0,Y 424.528,Z 609.326,A -85,B 0,C 180,E1 -9817.132,E2 -9817.132} C_VEL
LIN {X 0,Y 424.614,Z 603.288,A -85,B 0,C 180,E1 -9818.567,E2 -9818.567} C_VEL
LIN {X 0,Y 424.76,Z 595.781,A -85,B 0,C 180,E1 -9820.005,E2 -9820.005} C_VEL
LIN {X 0,Y 425.166,Z 586.43,A -85,B 0,C 180,E1 -9821.441,E2 -9821.441} C_VEL
LIN {X 0,Y 425.778,Z 575.909,A -85,B 0,C 180,E1 -9822.753,E2 -9822.753} C_VEL
LIN {X 0,Y 426.362,Z 565.225,A -85,B 0,C 180,E1 -9823.828,E2 -9823.828} C_VEL
LIN {X 0,Y 427.063,Z 553.5,A -85,B 0,C 180,E1 -9824.778,E2 -9824.778} C_VEL
LIN {X 0,Y 427.922,Z 540.456,A -85,B 0,C 180,E1 -9825.601,E2 -9825.601} C_VEL
LIN {X 0,Y 428.642,Z 527.266,A -85,B 0,C 180,E1 -9826.215,E2 -9826.215} C_VEL
LIN {X 0,Y 429.18,Z 513.74,A -85,B 0,C 180,E1 -9826.653,E2 -9826.653} C_VEL
LIN {X 0,Y 430.509,Z 438.648,A -85,B 0,C 180,E1 -9828.236,E2 -9828.236} C_VEL
LIN {X 0,Y 428.148,Z 413.974,A -85,B 0,C 180,E1 -9828.942,E2 -9828.942} C_VEL
LIN {X 0,Y 426.484,Z 401.654,A -85,B 0,C 180,E1 -9829.357,E2 -9829.357} C_VEL
LIN {X 0,Y 427.868,Z 377.127,A -85,B 0,C 180,E1 -9833.217,E2 -9833.217} C_VEL
LIN {X 0,Y 429.271,Z 357.103,A -85,B 0,C 180,E1 -9836.496,E2 -9836.496} C_VEL
LIN {X 0,Y 429.863,Z 348.232,A -85,B 0,C 180,E1 -9838.009,E2 -9838.009} C_VEL
LIN {X 0,Y 427.764,Z 337.871,A -85,B 0,C 180,E1 -9840.073,E2 -9840.073} C_VEL
LIN {X 0,Y 425.308,Z 328.513,A -85,B 0,C 180,E1 -9842.143,E2 -9842.143} C_VEL
LIN {X 0,Y 425.3,Z 328.509,A -85,B 0,C 180,E1 -9845.336,E2 -9845.336} C_VEL
LIN {X 0,Y 425.283,Z 328.512,A -85,B 0,C 180,E1 -9848.9,E2 -9848.9} C_VEL
LIN {X 0,Y 425.263,Z 328.514,A -85,B 0,C 180,E1 -9852.655,E2 -9852.655} C_VEL
LIN {X 0,Y 425.287,Z 328.509,A -85,B 0,C 180,E1 -9855.283,E2 -9855.283} C_VEL
LIN {X 0,Y 425.253,Z 328.514,A -85,B 0,C 180,E1 -9858.618,E2 -9858.618} C_VEL
LIN {X 0,Y 425.278,Z 328.508,A -85,B 0,C 180,E1 -9861.099,E2 -9861.099} C_VEL
LIN {X 0,Y 425.294,Z 328.507,A -85,B 0,C 180,E1 -9864.663,E2 -9864.663} C_VEL
LIN {X 0,Y 425.263,Z 328.514,A -85,B 0,C 180,E1 -9868.072,E2 -9868.072} C_VEL
LIN {X 0,Y 425.297,Z 328.51,A -85,B 0,C 180,E1 -9871.365,E2 -9871.365} C_VEL
LIN {X 0,Y 425.253,Z 328.514,A -85,B 0,C 180,E1 -9874.551,E2 -9874.551} C_VEL
LIN {X 0,Y 425.292,Z 328.513,A -85,B 0,C 180,E1 -9877.73,E2 -9877.73} C_VEL
LIN {X 0,Y 425.326,Z 328.506,A -85,B 0,C 180,E1 -9880.702,E2 -9880.702} C_VEL
LIN {X 0,Y 425.326,Z 328.507,A -85,B 0,C 180,E1 -9882.96,E2 -9882.96} C_VEL
LIN {X 0,Y 426.537,Z 331.661,A -85,B 0,C 180,E1 -9883.145,E2 -9883.145} C_VEL
LIN {X 0,Y 431.825,Z 343.897,A -85,B 0,C 180,E1 -9883.788,E2 -9883.788} C_VEL
LIN {X 0,Y 430.106,Z 418.82,A -85,B 0,C 180,E1 -9885.419,E2 -9885.419} C_VEL
LIN {X 0,Y 429.98,Z 432.057,A -85,B 0,C 180,E1 -9885.868,E2 -9885.868} C_VEL
LIN {X 0,Y 429.67,Z 445.212,A -85,B 0,C 180,E1 -9886.521,E2 -9886.521} C_VEL
LIN {X 0,Y 429.311,Z 455.985,A -85,B 0,C 180,E1 -9887.232,E2 -9887.232} C_VEL
LIN {X 0,Y 428.676,Z 467.254,A -85,B 0,C 180,E1 -9888.174,E2 -9888.174} C_VEL
LIN {X 0,Y 428.138,Z 477.41,A -85,B 0,C 180,E1 -9889.238,E2 -9889.238} C_VEL
LIN {X 0,Y 427.57,Z 485.735,A -85,B 0,C 180,E1 -9890.3,E2 -9890.3} C_VEL
LIN {X 0,Y 427.04,Z 493.381,A -85,B 0,C 180,E1 -9891.482,E2 -9891.482} C_VEL
LIN {X 0,Y 426.517,Z 500.807,A -85,B 0,C 180,E1 -9892.901,E2 -9892.901} C_VEL
LIN {X 0,Y 425.915,Z 506.76,A -85,B 0,C 180,E1 -9894.318,E2 -9894.318} C_VEL
LIN {X 0,Y 425.653,Z 511.388,A -85,B 0,C 180,E1 -9895.739,E2 -9895.739} C_VEL
LIN {X 0,Y 425.277,Z 514.914,A -85,B 0,C 180,E1 -9897.158,E2 -9897.158} C_VEL
LIN {X 0,Y 425.286,Z 516.667,A -85,B 0,C 180,E1 -9898.106,E2 -9898.106} C_VEL
LIN {X 0,Y 425.145,Z 517.983,A -85,B 0,C 180,E1 -9899.052,E2 -9899.052} C_VEL
LIN {X 0,Y 425.028,Z 518.867,A -85,B 0,C 180,E1 -9900,E2 -9900} C_VEL
LIN {X 0,Y 425.005,Z 519.342,A -85,B 0,C 180,E1 -9900.947,E2 -9900.947} C_VEL
LIN {X 0,Y 424.758,Z 519.435,A -85,B 0,C 180,E1 -9901.896,E2 -9901.896} C_VEL
LIN {X 0,Y 424.779,Z 519.044,A -85,B 0,C 180,E1 -9902.845,E2 -9902.845} C_VEL
LIN {X 0,Y 424.863,Z 518.249,A -85,B 0,C 180,E1 -9903.793,E2 -9903.793} C_VEL
LIN {X 0,Y 425.034,Z 517.046,A -85,B 0,C 180,E1 -9904.742,E2 -9904.742} C_VEL
LIN {X 0,Y 425.128,Z 514.42,A -85,B 0,C 180,E1 -9906.168,E2 -9906.168} C_VEL
LIN {X 0,Y 425.272,Z 510.759,A -85,B 0,C 180,E1 -9907.597,E2 -9907.597} C_VEL
LIN {X 0,Y 425.446,Z 505.955,A -85,B 0,C 180,E1 -9909.028,E2 -9909.028} C_VEL
LIN {X 0,Y 425.736,Z 499.832,A -85,B 0,C 180,E1 -9910.462,E2 -9910.462} C_VEL
LIN {X 0,Y 426.138,Z 492.182,A -85,B 0,C 180,E1 -9911.897,E2 -9911.897} C_VEL
LIN {X 0,Y 426.549,Z 484.374,A -85,B 0,C 180,E1 -9913.094,E2 -9913.094} C_VEL
LIN {X 0,Y 426.956,Z 474.89,A -85,B 0,C 180,E1 -9914.294,E2 -9914.294} C_VEL
LIN {X 0,Y 427.521,Z 464.292,A -85,B 0,C 180,E1 -9915.371,E2 -9915.371} C_VEL
LIN {X 0,Y 427.909,Z 452.533,A -85,B 0,C 180,E1 -9916.335,E2 -9916.335} C_VEL
LIN {X 0,Y 428.396,Z 440.172,A -85,B 0,C 180,E1 -9917.113,E2 -9917.113} C_VEL
LIN {X 0,Y 428.648,Z 426.635,A -85,B 0,C 180,E1 -9917.746,E2 -9917.746} C_VEL
LIN {X 0,Y 428.758,Z 414.003,A -85,B 0,C 180,E1 -9918.145,E2 -9918.145} C_VEL
LIN {X 0,Y 429.779,Z 341.76,A -85,B 0,C 180,E1 -9919.569,E2 -9919.569} C_VEL
LIN {X 0,Y 425.341,Z 328.503,A -85,B 0,C 180,E1 -9920.032,E2 -9920.032} C_VEL
LIN {X 0,Y 425.307,Z 328.505,A -85,B 0,C 180,E1 -9923.365,E2 -9923.365} C_VEL
LIN {X 0,Y 425.348,Z 328.504,A -85,B 0,C 180,E1 -9926.844,E2 -9926.844} C_VEL
LIN {X 0,Y 425.291,Z 328.506,A -85,B 0,C 180,E1 -9929.719,E2 -9929.719} C_VEL
LIN {X 0,Y 425.281,Z 328.51,A -85,B 0,C 180,E1 -9933.048,E2 -9933.048} C_VEL
LIN {X 0,Y 425.28,Z 328.508,A -85,B 0,C 180,E1 -9935.928,E2 -9935.928} C_VEL
LIN {X 0,Y 425.28,Z 328.51,A -85,B 0,C 180,E1 -9939.04,E2 -9939.04} C_VEL
LIN {X 0,Y 425.288,Z 328.507,A -85,B 0,C 180,E1 -9941.958,E2 -9941.958} C_VEL
LIN {X 0,Y 425.283,Z 328.508,A -85,B 0,C 180,E1 -9945.283,E2 -9945.283} C_VEL
LIN {X 0,Y 425.273,Z 328.514,A -85,B 0,C 180,E1 -9948.621,E2 -9948.621} C_VEL
LIN {X 0,Y 425.314,Z 328.504,A -85,B 0,C 180,E1 -9951.103,E2 -9951.103} C_VEL
LIN {X 0,Y 425.298,Z 328.509,A -85,B 0,C 180,E1 -9954.664,E2 -9954.664} C_VEL
LIN {X 0,Y 425.263,Z 328.512,A -85,B 0,C 180,E1 -9958.073,E2 -9958.073} C_VEL
LIN {X 0,Y 425.329,Z 328.502,A -85,B 0,C 180,E1 -9961.368,E2 -9961.368} C_VEL
LIN {X 0,Y 425.294,Z 328.51,A -85,B 0,C 180,E1 -9964.555,E2 -9964.555} C_VEL
LIN {X 0,Y 425.285,Z 328.508,A -85,B 0,C 180,E1 -9967.661,E2 -9967.661} C_VEL
LIN {X 0,Y 425.359,Z 328.5,A -85,B 0,C 180,E1 -9970.704,E2 -9970.704} C_VEL
LIN {X 0,Y 425.386,Z 328.495,A -85,B 0,C 180,E1 -9973.688,E2 -9973.688} C_VEL
LIN {X 0,Y 425.409,Z 328.492,A -85,B 0,C 180,E1 -9977.598,E2 -9977.598} C_VEL
LIN {X 0,Y 425.44,Z 328.488,A -85,B 0,C 180,E1 -9981.45,E2 -9981.45} C_VEL
LIN {X 0,Y 425.552,Z 328.479,A -85,B 0,C 180,E1 -9984.313,E2 -9984.313} C_VEL
LIN {X 0,Y 425.549,Z 328.474,A -85,B 0,C 180,E1 -9987.331,E2 -9987.331} C_VEL
LIN {X 0,Y 424.871,Z 328.563,A -85,B 0,C 180,E1 -9988.122,E2 -9988.122} C_VEL
LIN {X 0,Y 421.997,Z 328.917,A -85,B 0,C 180,E1 -9989.408,E2 -9989.408} C_VEL
LIN {X 0,Y 419.586,Z 329.22,A -85,B 0,C 180,E1 -9990.447,E2 -9990.447} C_VEL
LIN {X 0,Y 418.578,Z 329.343,A -85,B 0,C 180,E1 -9991.249,E2 -9991.249} C_VEL
LIN {X 0,Y 418.51,Z 329.351,A -85,B 0,C 180,E1 -9991.521,E2 -9991.521} C_VEL
LIN {X 0,Y 418.508,Z 329.352,A -85,B 0,C 180,E1 -9992.888,E2 -9992.888} C_VEL
LIN {X 0,Y 418.491,Z 329.354,A -85,B 0,C 180,E1 -9996.751,E2 -9996.751} C_VEL
LIN {X 0,Y 418.339,Z 329.374,A -85,B 0,C 180,E1 -9999.672,E2 -9999.672} C_VEL
LIN {X 0,Y 418.344,Z 329.373,A -85,B 0,C 180,E1 -10003.001,E2 -10003.001} C_VEL
LIN {X 0,Y 418.311,Z 329.377,A -85,B 0,C 180,E1 -10006.736,E2 -10006.736} C_VEL
LIN {X 0,Y 418.269,Z 329.384,A -85,B 0,C 180,E1 -10009.791,E2 -10009.791} C_VEL
LIN {X 0,Y 418.237,Z 329.386,A -85,B 0,C 180,E1 -10012.737,E2 -10012.737} C_VEL
LIN {X 0,Y 418.27,Z 329.386,A -85,B 0,C 180,E1 -10015.904,E2 -10015.904} C_VEL
LIN {X 0,Y 418.263,Z 329.383,A -85,B 0,C 180,E1 -10019.162,E2 -10019.162} C_VEL
LIN {X 0,Y 418.256,Z 329.384,A -85,B 0,C 180,E1 -10022.845,E2 -10022.845} C_VEL
LIN {X 0,Y 418.248,Z 329.386,A -85,B 0,C 180,E1 -10026.239,E2 -10026.239} C_VEL
LIN {X 0,Y 418.255,Z 329.386,A -85,B 0,C 180,E1 -10029.682,E2 -10029.682} C_VEL
LIN {X 0,Y 418.229,Z 329.388,A -85,B 0,C 180,E1 -10032.322,E2 -10032.322} C_VEL
LIN {X 0,Y 418.235,Z 329.386,A -85,B 0,C 180,E1 -10035.109,E2 -10035.109} C_VEL
LIN {X 0,Y 418.24,Z 329.39,A -85,B 0,C 180,E1 -10037.768,E2 -10037.768} C_VEL
LIN {X 0,Y 418.246,Z 329.385,A -85,B 0,C 180,E1 -10040.621,E2 -10040.621} C_VEL
LIN {X 0,Y 418.243,Z 329.388,A -85,B 0,C 180,E1 -10043.976,E2 -10043.976} C_VEL
LIN {X 0,Y 418.258,Z 329.384,A -85,B 0,C 180,E1 -10047.157,E2 -10047.157} C_VEL
LIN {X 0,Y 418.27,Z 329.382,A -85,B 0,C 180,E1 -10050.896,E2 -10050.896} C_VEL
LIN {X 0,Y 418.33,Z 329.376,A -85,B 0,C 180,E1 -10053.799,E2 -10053.799} C_VEL
LIN {X 0,Y 422.971,Z 343.296,A -85,B 0,C 180,E1 -10054.278,E2 -10054.278} C_VEL
LIN {X 0,Y 421.925,Z 417.033,A -85,B 0,C 180,E1 -10055.752,E2 -10055.752} C_VEL
LIN {X 0,Y 421.834,Z 428.429,A -85,B 0,C 180,E1 -10056.138,E2 -10056.138} C_VEL
LIN {X 0,Y 421.504,Z 441.18,A -85,B 0,C 180,E1 -10056.752,E2 -10056.752} C_VEL
LIN {X 0,Y 421.074,Z 453.612,A -85,B 0,C 180,E1 -10057.555,E2 -10057.555} C_VEL
LIN {X 0,Y 420.621,Z 464.276,A -85,B 0,C 180,E1 -10058.433,E2 -10058.433} C_VEL
LIN {X 0,Y 420.129,Z 474.819,A -85,B 0,C 180,E1 -10059.519,E2 -10059.519} C_VEL
LIN {X 0,Y 419.595,Z 484.087,A -85,B 0,C 180,E1 -10060.683,E2 -10060.683} C_VEL
LIN {X 0,Y 419.171,Z 492.261,A -85,B 0,C 180,E1 -10061.93,E2 -10061.93} C_VEL
LIN {X 0,Y 418.746,Z 500.134,A -85,B 0,C 180,E1 -10063.423,E2 -10063.423} C_VEL
LIN {X 0,Y 418.397,Z 506.413,A -85,B 0,C 180,E1 -10064.909,E2 -10064.909} C_VEL
LIN {X 0,Y 418.13,Z 511.345,A -85,B 0,C 180,E1 -10066.39,E2 -10066.39} C_VEL
LIN {X 0,Y 418.015,Z 515.066,A -85,B 0,C 180,E1 -10067.869,E2 -10067.869} C_VEL
LIN {X 0,Y 417.849,Z 517.711,A -85,B 0,C 180,E1 -10069.339,E2 -10069.339} C_VEL
LIN {X 0,Y 417.841,Z 518.885,A -85,B 0,C 180,E1 -10070.317,E2 -10070.317} C_VEL
LIN {X 0,Y 417.862,Z 519.654,A -85,B 0,C 180,E1 -10071.294,E2 -10071.294} C_VEL
LIN {X 0,Y 417.968,Z 519.999,A -85,B 0,C 180,E1 -10072.783,E2 -10072.783} C_VEL
LIN {X 0,Y 418.007,Z 519.405,A -85,B 0,C 180,E1 -10074.211,E2 -10074.211} C_VEL
LIN {X 0,Y 418.05,Z 518.507,A -85,B 0,C 180,E1 -10075.179,E2 -10075.179} C_VEL
LIN {X 0,Y 418.129,Z 517.138,A -85,B 0,C 180,E1 -10076.145,E2 -10076.145} C_VEL
LIN {X 0,Y 418.446,Z 514.253,A -85,B 0,C 180,E1 -10077.594,E2 -10077.594} C_VEL
LIN {X 0,Y 418.781,Z 510.305,A -85,B 0,C 180,E1 -10079.039,E2 -10079.039} C_VEL
LIN {X 0,Y 419.209,Z 505.182,A -85,B 0,C 180,E1 -10080.481,E2 -10080.481} C_VEL
LIN {X 0,Y 419.74,Z 498.746,A -85,B 0,C 180,E1 -10081.919,E2 -10081.919} C_VEL
LIN {X 0,Y 420.413,Z 490.656,A -85,B 0,C 180,E1 -10083.355,E2 -10083.355} C_VEL
LIN {X 0,Y 420.995,Z 482.37,A -85,B 0,C 180,E1 -10084.549,E2 -10084.549} C_VEL
LIN {X 0,Y 421.675,Z 472.203,A -85,B 0,C 180,E1 -10085.74,E2 -10085.74} C_VEL
LIN {X 0,Y 422.159,Z 462.101,A -85,B 0,C 180,E1 -10086.693,E2 -10086.693} C_VEL
LIN {X 0,Y 422.728,Z 450.985,A -85,B 0,C 180,E1 -10087.523,E2 -10087.523} C_VEL
LIN {X 0,Y 423.09,Z 438.707,A -85,B 0,C 180,E1 -10088.238,E2 -10088.238} C_VEL
LIN {X 0,Y 423.328,Z 424.876,A -85,B 0,C 180,E1 -10088.804,E2 -10088.804} C_VEL
LIN {X 0,Y 423.477,Z 409.519,A -85,B 0,C 180,E1 -10089.192,E2 -10089.192} C_VEL
LIN {X 0,Y 425.037,Z 345.391,A -85,B 0,C 180,E1 -10090.556,E2 -10090.556} C_VEL
LIN {X 0,Y 419.294,Z 332.192,A -85,B 0,C 180,E1 -10091.239,E2 -10091.239} C_VEL
LIN {X 0,Y 418.302,Z 329.382,A -85,B 0,C 180,E1 -10091.396,E2 -10091.396} C_VEL
LIN {X 0,Y 418.305,Z 329.379,A -85,B 0,C 180,E1 -10093.605,E2 -10093.605} C_VEL
LIN {X 0,Y 418.31,Z 329.381,A -85,B 0,C 180,E1 -10096.732,E2 -10096.732} C_VEL
LIN {X 0,Y 418.241,Z 329.391,A -85,B 0,C 180,E1 -10099.777,E2 -10099.777} C_VEL
LIN {X 0,Y 418.228,Z 329.388,A -85,B 0,C 180,E1 -10102.737,E2 -10102.737} C_VEL
LIN {X 0,Y 418.214,Z 329.394,A -85,B 0,C 180,E1 -10105.908,E2 -10105.908} C_VEL
LIN {X 0,Y 418.26,Z 329.383,A -85,B 0,C 180,E1 -10109.163,E2 -10109.163} C_VEL
LIN {X 0,Y 418.255,Z 329.383,A -85,B 0,C 180,E1 -10112.842,E2 -10112.842} C_VEL
LIN {X 0,Y 418.243,Z 329.385,A -85,B 0,C 180,E1 -10116.237,E2 -10116.237} C_VEL
LIN {X 0,Y 418.202,Z 329.389,A -85,B 0,C 180,E1 -10119.688,E2 -10119.688} C_VEL
LIN {X 0,Y 418.211,Z 329.388,A -85,B 0,C 180,E1 -10122.318,E2 -10122.318} C_VEL
LIN {X 0,Y 418.238,Z 329.386,A -85,B 0,C 180,E1 -10125.108,E2 -10125.108} C_VEL
LIN {X 0,Y 418.227,Z 329.391,A -85,B 0,C 180,E1 -10127.765,E2 -10127.765} C_VEL
LIN {X 0,Y 418.241,Z 329.389,A -85,B 0,C 180,E1 -10131.556,E2 -10131.556} C_VEL
LIN {X 0,Y 418.261,Z 329.386,A -85,B 0,C 180,E1 -10135.159,E2 -10135.159} C_VEL
LIN {X 0,Y 418.29,Z 329.561,A -85,B 0,C 180,E1 -10138.54,E2 -10138.54} C_VEL
LIN {X 0,Y 421.822,Z 345.314,A -85,B 0,C 180,E1 -10141.32,E2 -10141.32} C_VEL
LIN {X 0,Y 422.77,Z 350.84,A -85,B 0,C 180,E1 -10142.259,E2 -10142.259} C_VEL
LIN {X 0,Y 421.252,Z 373.856,A -85,B 0,C 180,E1 -10145.873,E2 -10145.873} C_VEL
LIN {X 0,Y 419.875,Z 398.642,A -85,B 0,C 180,E1 -10149.723,E2 -10149.723} C_VEL
LIN {X 0,Y 419.536,Z 405.429,A -85,B 0,C 180,E1 -10150.757,E2 -10150.757} C_VEL
LIN {X 0,Y 421.998,Z 427.036,A -85,B 0,C 180,E1 -10151.405,E2 -10151.405} C_VEL
LIN {X 0,Y 423.234,Z 441.78,A -85,B 0,C 180,E1 -10151.808,E2 -10151.808} C_VEL
LIN {X 0,Y 421.8,Z 515.819,A -85,B 0,C 180,E1 -10153.39,E2 -10153.39} C_VEL
LIN {X 0,Y 421.272,Z 528.605,A -85,B 0,C 180,E1 -10153.835,E2 -10153.835} C_VEL
LIN {X 0,Y 420.515,Z 541.643,A -85,B 0,C 180,E1 -10154.49,E2 -10154.49} C_VEL
LIN {X 0,Y 419.697,Z 555.969,A -85,B 0,C 180,E1 -10155.452,E2 -10155.452} C_VEL
LIN {X 0,Y 419.027,Z 567.52,A -85,B 0,C 180,E1 -10156.419,E2 -10156.419} C_VEL
LIN {X 0,Y 418.721,Z 575.6,A -85,B 0,C 180,E1 -10157.246,E2 -10157.246} C_VEL
LIN {X 0,Y 418.11,Z 584.76,A -85,B 0,C 180,E1 -10158.363,E2 -10158.363} C_VEL
LIN {X 0,Y 417.78,Z 593.004,A -85,B 0,C 180,E1 -10159.581,E2 -10159.581} C_VEL
LIN {X 0,Y 417.522,Z 601.054,A -85,B 0,C 180,E1 -10161.042,E2 -10161.042} C_VEL
LIN {X 0,Y 417.436,Z 606.517,A -85,B 0,C 180,E1 -10162.259,E2 -10162.259} C_VEL
LIN {X 0,Y 417.453,Z 611.758,A -85,B 0,C 180,E1 -10163.709,E2 -10163.709} C_VEL
LIN {X 0,Y 417.491,Z 615.81,A -85,B 0,C 180,E1 -10165.172,E2 -10165.172} C_VEL
LIN {X 0,Y 417.65,Z 617.866,A -85,B 0,C 180,E1 -10166.14,E2 -10166.14} C_VEL
LIN {X 0,Y 417.545,Z 619.435,A -85,B 0,C 180,E1 -10167.105,E2 -10167.105} C_VEL
LIN {X 0,Y 417.511,Z 620.555,A -85,B 0,C 180,E1 -10168.071,E2 -10168.071} C_VEL
LIN {X 0,Y 417.529,Z 621.203,A -85,B 0,C 180,E1 -10169.035,E2 -10169.035} C_VEL
LIN {X 0,Y 417.564,Z 621.425,A -85,B 0,C 180,E1 -10170,E2 -10170} C_VEL
LIN {X 0,Y 417.527,Z 621.211,A -85,B 0,C 180,E1 -10170.964,E2 -10170.964} C_VEL
LIN {X 0,Y 417.51,Z 620.529,A -85,B 0,C 180,E1 -10171.929,E2 -10171.929} C_VEL
LIN {X 0,Y 417.551,Z 619.404,A -85,B 0,C 180,E1 -10172.894,E2 -10172.894} C_VEL
LIN {X 0,Y 417.541,Z 616.879,A -85,B 0,C 180,E1 -10174.344,E2 -10174.344} C_VEL
LIN {X 0,Y 417.476,Z 613.273,A -85,B 0,C 180,E1 -10175.797,E2 -10175.797} C_VEL
LIN {X 0,Y 417.449,Z 608.51,A -85,B 0,C 180,E1 -10177.254,E2 -10177.254} C_VEL
LIN {X 0,Y 417.512,Z 602.472,A -85,B 0,C 180,E1 -10178.714,E2 -10178.714} C_VEL
LIN {X 0,Y 417.698,Z 594.994,A -85,B 0,C 180,E1 -10180.176,E2 -10180.176} C_VEL
LIN {X 0,Y 418.135,Z 585.701,A -85,B 0,C 180,E1 -10181.636,E2 -10181.636} C_VEL
LIN {X 0,Y 418.752,Z 575.724,A -85,B 0,C 180,E1 -10182.909,E2 -10182.909} C_VEL
LIN {X 0,Y 419.377,Z 564.637,A -85,B 0,C 180,E1 -10184.063,E2 -10184.063} C_VEL
LIN {X 0,Y 420.186,Z 553.036,A -85,B 0,C 180,E1 -10185.026,E2 -10185.026} C_VEL
LIN {X 0,Y 421.064,Z 540.209,A -85,B 0,C 180,E1 -10185.862,E2 -10185.862} C_VEL
LIN {X 0,Y 421.842,Z 527.387,A -85,B 0,C 180,E1 -10186.484,E2 -10186.484} C_VEL
LIN {X 0,Y 422.459,Z 513.488,A -85,B 0,C 180,E1 -10186.957,E2 -10186.957} C_VEL
LIN {X 0,Y 423.952,Z 439.824,A -85,B 0,C 180,E1 -10188.562,E2 -10188.562} C_VEL
LIN {X 0,Y 421.649,Z 415.066,A -85,B 0,C 180,E1 -10189.296,E2 -10189.296} C_VEL
LIN {X 0,Y 419.638,Z 400.385,A -85,B 0,C 180,E1 -10189.81,E2 -10189.81} C_VEL
LIN {X 0,Y 420.94,Z 378.587,A -85,B 0,C 180,E1 -10193.323,E2 -10193.323} C_VEL
LIN {X 0,Y 422.48,Z 358.527,A -85,B 0,C 180,E1 -10196.689,E2 -10196.689} C_VEL
LIN {X 0,Y 423.152,Z 350.559,A -85,B 0,C 180,E1 -10198.074,E2 -10198.074} C_VEL
LIN {X 0,Y 421.293,Z 340.944,A -85,B 0,C 180,E1 -10200.03,E2 -10200.03} C_VEL
LIN {X 0,Y 418.238,Z 329.402,A -85,B 0,C 180,E1 -10202.669,E2 -10202.669} C_VEL
LIN {X 0,Y 418.26,Z 329.386,A -85,B 0,C 180,E1 -10204.841,E2 -10204.841} C_VEL
LIN {X 0,Y 418.24,Z 329.391,A -85,B 0,C 180,E1 -10208.443,E2 -10208.443} C_VEL
LIN {X 0,Y 418.225,Z 329.393,A -85,B 0,C 180,E1 -10212.235,E2 -10212.235} C_VEL
LIN {X 0,Y 418.238,Z 329.387,A -85,B 0,C 180,E1 -10215.108,E2 -10215.108} C_VEL
LIN {X 0,Y 418.225,Z 329.391,A -85,B 0,C 180,E1 -10217.764,E2 -10217.764} C_VEL
LIN {X 0,Y 418.236,Z 329.388,A -85,B 0,C 180,E1 -10221.556,E2 -10221.556} C_VEL
LIN {X 0,Y 418.251,Z 329.384,A -85,B 0,C 180,E1 -10225.158,E2 -10225.158} C_VEL
LIN {X 0,Y 418.244,Z 329.387,A -85,B 0,C 180,E1 -10227.471,E2 -10227.471} C_VEL
LIN {X 0,Y 418.261,Z 329.384,A -85,B 0,C 180,E1 -10230.898,E2 -10230.898} C_VEL
LIN {X 0,Y 418.212,Z 329.394,A -85,B 0,C 180,E1 -10234.092,E2 -10234.092} C_VEL
LIN {X 0,Y 418.226,Z 329.392,A -85,B 0,C 180,E1 -10237.263,E2 -10237.263} C_VEL
LIN {X 0,Y 418.252,Z 329.387,A -85,B 0,C 180,E1 -10240.362,E2 -10240.362} C_VEL
LIN {X 0,Y 418.286,Z 329.411,A -85,B 0,C 180,E1 -10242.508,E2 -10242.508} C_VEL
LIN {X 0,Y 419.364,Z 332.37,A -85,B 0,C 180,E1 -10242.666,E2 -10242.666} C_VEL
LIN {X 0,Y 424.684,Z 344.002,A -85,B 0,C 180,E1 -10243.336,E2 -10243.336} C_VEL
LIN {X 0,Y 425.389,Z 346.307,A -85,B 0,C 180,E1 -10243.441,E2 -10243.441} C_VEL
LIN {X 0,Y 423.522,Z 418.756,A -85,B 0,C 180,E1 -10245.064,E2 -10245.064} C_VEL
LIN {X 0,Y 423.409,Z 431.675,A -85,B 0,C 180,E1 -10245.49,E2 -10245.49} C_VEL
LIN {X 0,Y 423.068,Z 444.603,A -85,B 0,C 180,E1 -10246.123,E2 -10246.123} C_VEL
LIN {X 0,Y 422.647,Z 456.515,A -85,B 0,C 180,E1 -10246.905,E2 -10246.905} C_VEL
LIN {X 0,Y 422.006,Z 467.891,A -85,B 0,C 180,E1 -10247.862,E2 -10247.862} C_VEL
LIN {X 0,Y 421.412,Z 478.091,A -85,B 0,C 180,E1 -10248.942,E2 -10248.942} C_VEL
LIN {X 0,Y 420.735,Z 487.482,A -85,B 0,C 180,E1 -10250.165,E2 -10250.165} C_VEL
LIN {X 0,Y 420.063,Z 496.157,A -85,B 0,C 180,E1 -10251.581,E2 -10251.581} C_VEL
LIN {X 0,Y 419.606,Z 502.163,A -85,B 0,C 180,E1 -10252.783,E2 -10252.783} C_VEL
LIN {X 0,Y 418.966,Z 508.035,A -85,B 0,C 180,E1 -10254.223,E2 -10254.223} C_VEL
LIN {X 0,Y 418.675,Z 512.587,A -85,B 0,C 180,E1 -10255.667,E2 -10255.667} C_VEL
LIN {X 0,Y 418.305,Z 516.041,A -85,B 0,C 180,E1 -10257.11,E2 -10257.11} C_VEL
LIN {X 0,Y 418.279,Z 517.755,A -85,B 0,C 180,E1 -10258.074,E2 -10258.074} C_VEL
LIN {X 0,Y 418.138,Z 519.01,A -85,B 0,C 180,E1 -10259.036,E2 -10259.036} C_VEL
LIN {X 0,Y 418,Z 519.858,A -85,B 0,C 180,E1 -10260,E2 -10260} C_VEL
LIN {X 0,Y 417.973,Z 520.294,A -85,B 0,C 180,E1 -10260.963,E2 -10260.963} C_VEL
LIN {X 0,Y 417.715,Z 520.32,A -85,B 0,C 180,E1 -10261.928,E2 -10261.928} C_VEL
LIN {X 0,Y 417.735,Z 519.884,A -85,B 0,C 180,E1 -10262.893,E2 -10262.893} C_VEL
LIN {X 0,Y 417.83,Z 519.046,A -85,B 0,C 180,E1 -10263.857,E2 -10263.857} C_VEL
LIN {X 0,Y 418.013,Z 517.786,A -85,B 0,C 180,E1 -10264.822,E2 -10264.822} C_VEL
LIN {X 0,Y 418.101,Z 515.078,A -85,B 0,C 180,E1 -10266.272,E2 -10266.272} C_VEL
LIN {X 0,Y 418.234,Z 511.318,A -85,B 0,C 180,E1 -10267.725,E2 -10267.725} C_VEL
LIN {X 0,Y 418.428,Z 506.39,A -85,B 0,C 180,E1 -10269.181,E2 -10269.181} C_VEL
LIN {X 0,Y 418.725,Z 500.145,A -85,B 0,C 180,E1 -10270.639,E2 -10270.639} C_VEL
LIN {X 0,Y 419.158,Z 492.357,A -85,B 0,C 180,E1 -10272.098,E2 -10272.098} C_VEL
LIN {X 0,Y 419.601,Z 484.399,A -85,B 0,C 180,E1 -10273.314,E2 -10273.314} C_VEL
LIN {X 0,Y 420.023,Z 474.656,A -85,B 0,C 180,E1 -10274.535,E2 -10274.535} C_VEL
LIN {X 0,Y 420.57,Z 463.821,A -85,B 0,C 180,E1 -10275.632,E2 -10275.632} C_VEL
LIN {X 0,Y 420.945,Z 453.385,A -85,B 0,C 180,E1 -10276.488,E2 -10276.488} C_VEL
LIN {X 0,Y 421.443,Z 441.047,A -85,B 0,C 180,E1 -10277.28,E2 -10277.28} C_VEL
LIN {X 0,Y 421.738,Z 427.556,A -85,B 0,C 180,E1 -10277.921,E2 -10277.921} C_VEL
LIN {X 0,Y 421.852,Z 415.179,A -85,B 0,C 180,E1 -10278.326,E2 -10278.326} C_VEL
LIN {X 0,Y 422.855,Z 343.059,A -85,B 0,C 180,E1 -10279.789,E2 -10279.789} C_VEL
LIN {X 0,Y 418.286,Z 329.383,A -85,B 0,C 180,E1 -10280.269,E2 -10280.269} C_VEL
LIN {X 0,Y 418.288,Z 329.379,A -85,B 0,C 180,E1 -10283.781,E2 -10283.781} C_VEL
LIN {X 0,Y 418.31,Z 329.378,A -85,B 0,C 180,E1 -10287.07,E2 -10287.07} C_VEL
LIN {X 0,Y 418.244,Z 329.385,A -85,B 0,C 180,E1 -10290.272,E2 -10290.272} C_VEL
LIN {X 0,Y 418.247,Z 329.384,A -85,B 0,C 180,E1 -10293.677,E2 -10293.677} C_VEL
LIN {X 0,Y 418.238,Z 329.386,A -85,B 0,C 180,E1 -10297.224,E2 -10297.224} C_VEL
LIN {X 0,Y 418.243,Z 329.384,A -85,B 0,C 180,E1 -10299.682,E2 -10299.682} C_VEL
LIN {X 0,Y 418.228,Z 329.389,A -85,B 0,C 180,E1 -10302.321,E2 -10302.321} C_VEL
LIN {X 0,Y 418.234,Z 329.387,A -85,B 0,C 180,E1 -10305.108,E2 -10305.108} C_VEL
LIN {X 0,Y 418.238,Z 329.385,A -85,B 0,C 180,E1 -10307.766,E2 -10307.766} C_VEL
LIN {X 0,Y 418.258,Z 329.387,A -85,B 0,C 180,E1 -10310.618,E2 -10310.618} C_VEL
LIN {X 0,Y 418.244,Z 329.385,A -85,B 0,C 180,E1 -10313.976,E2 -10313.976} C_VEL
LIN {X 0,Y 418.255,Z 329.383,A -85,B 0,C 180,E1 -10317.156,E2 -10317.156} C_VEL
LIN {X 0,Y 418.266,Z 329.383,A -85,B 0,C 180,E1 -10320.895,E2 -10320.895} C_VEL
LIN {X 0,Y 418.269,Z 329.383,A -85,B 0,C 180,E1 -10324.096,E2 -10324.096} C_VEL
LIN {X 0,Y 418.236,Z 329.386,A -85,B 0,C 180,E1 -10327.264,E2 -10327.264} C_VEL
LIN {X 0,Y 418.281,Z 329.385,A -85,B 0,C 180,E1 -10330.364,E2 -10330.364} C_VEL
LIN {X 0,Y 418.314,Z 329.376,A -85,B 0,C 180,E1 -10333.405,E2 -10333.405} C_VEL
LIN {X 0,Y 418.343,Z 329.373,A -85,B 0,C 180,E1 -10336.999,E2 -10336.999} C_VEL
LIN {X 0,Y 418.354,Z 329.376,A -85,B 0,C 180,E1 -10340.329,E2 -10340.329} C_VEL
LIN {X 0,Y 418.491,Z 329.354,A -85,B 0,C 180,E1 -10343.249,E2 -10343.249} C_VEL
LIN {X 0,Y 418.337,Z 329.373,A -85,B 0,C 180,E1 -10345.182,E2 -10345.182} C_VEL
LIN {X 0,Y 418.542,Z 329.351,A -85,B 0,C 180,E1 -10348.076,E2 -10348.076} C_VEL
LIN {X 0,Y 418.67,Z 329.334,A -85,B 0,C 180,E1 -10350,E2 -10350} C_VEL
LIN {X 0,Y 418.51,Z 329.351,A -85,B 0,C 180,E1 -10351.521,E2 -10351.521} C_VEL
LIN {X 0,Y 417.847,Z 329.438,A -85,B 0,C 180,E1 -10352.323,E2 -10352.323} C_VEL
LIN {X 0,Y 414.898,Z 329.802,A -85,B 0,C 180,E1 -10353.624,E2 -10353.624} C_VEL
LIN {X 0,Y 412.445,Z 330.108,A -85,B 0,C 180,E1 -10354.674,E2 -10354.674} C_VEL
LIN {X 0,Y 411.478,Z 330.228,A -85,B 0,C 180,E1 -10355.488,E2 -10355.488} C_VEL
LIN {X 0,Y 411.446,Z 330.233,A -85,B 0,C 180,E1 -10355.763,E2 -10355.763} C_VEL
LIN {X 0,Y 411.479,Z 330.229,A -85,B 0,C 180,E1 -10357.854,E2 -10357.854} C_VEL
LIN {X 0,Y 411.282,Z 330.254,A -85,B 0,C 180,E1 -10361.833,E2 -10361.833} C_VEL
LIN {X 0,Y 411.258,Z 330.255,A -85,B 0,C 180,E1 -10364.853,E2 -10364.853} C_VEL
LIN {X 0,Y 411.251,Z 330.259,A -85,B 0,C 180,E1 -10367.915,E2 -10367.915} C_VEL
LIN {X 0,Y 411.195,Z 330.263,A -85,B 0,C 180,E1 -10371.034,E2 -10371.034} C_VEL
LIN {X 0,Y 411.226,Z 330.262,A -85,B 0,C 180,E1 -10374.216,E2 -10374.216} C_VEL
LIN {X 0,Y 411.257,Z 330.256,A -85,B 0,C 180,E1 -10377.478,E2 -10377.478} C_VEL
LIN {X 0,Y 411.188,Z 330.264,A -85,B 0,C 180,E1 -10380.848,E2 -10380.848} C_VEL
LIN {X 0,Y 411.205,Z 330.263,A -85,B 0,C 180,E1 -10384.334,E2 -10384.334} C_VEL
LIN {X 0,Y 411.201,Z 330.266,A -85,B 0,C 180,E1 -10387.974,E2 -10387.974} C_VEL
LIN {X 0,Y 411.183,Z 330.265,A -85,B 0,C 180,E1 -10390.505,E2 -10390.505} C_VEL
LIN {X 0,Y 411.173,Z 330.266,A -85,B 0,C 180,E1 -10393.134,E2 -10393.134} C_VEL
LIN {X 0,Y 411.168,Z 330.271,A -85,B 0,C 180,E1 -10395.882,E2 -10395.882} C_VEL
LIN {X 0,Y 411.164,Z 330.267,A -85,B 0,C 180,E1 -10398.772,E2 -10398.772} C_VEL
LIN {X 0,Y 411.192,Z 330.266,A -85,B 0,C 180,E1 -10402.027,E2 -10402.027} C_VEL
LIN {X 0,Y 411.206,Z 330.266,A -85,B 0,C 180,E1 -10405.667,E2 -10405.667} C_VEL
LIN {X 0,Y 411.191,Z 330.264,A -85,B 0,C 180,E1 -10409.153,E2 -10409.153} C_VEL
LIN {X 0,Y 411.261,Z 330.256,A -85,B 0,C 180,E1 -10412.523,E2 -10412.523} C_VEL
LIN {X 0,Y 411.285,Z 330.254,A -85,B 0,C 180,E1 -10413.555,E2 -10413.555} C_VEL
LIN {X 0,Y 416.12,Z 344.783,A -85,B 0,C 180,E1 -10414.059,E2 -10414.059} C_VEL
LIN {X 0,Y 415.023,Z 417.83,A -85,B 0,C 180,E1 -10415.555,E2 -10415.555} C_VEL
LIN {X 0,Y 414.933,Z 429.209,A -85,B 0,C 180,E1 -10415.949,E2 -10415.949} C_VEL
LIN {X 0,Y 414.622,Z 440.839,A -85,B 0,C 180,E1 -10416.507,E2 -10416.507} C_VEL
LIN {X 0,Y 414.187,Z 453.078,A -85,B 0,C 180,E1 -10417.293,E2 -10417.293} C_VEL
LIN {X 0,Y 413.698,Z 464.009,A -85,B 0,C 180,E1 -10418.185,E2 -10418.185} C_VEL
LIN {X 0,Y 413.181,Z 475.018,A -85,B 0,C 180,E1 -10419.314,E2 -10419.314} C_VEL
LIN {X 0,Y 412.578,Z 485.146,A -85,B 0,C 180,E1 -10420.6,E2 -10420.6} C_VEL
LIN {X 0,Y 412.149,Z 493.289,A -85,B 0,C 180,E1 -10421.869,E2 -10421.869} C_VEL
LIN {X 0,Y 411.72,Z 501.136,A -85,B 0,C 180,E1 -10423.387,E2 -10423.387} C_VEL
LIN {X 0,Y 411.395,Z 506.452,A -85,B 0,C 180,E1 -10424.646,E2 -10424.646} C_VEL
LIN {X 0,Y 411.113,Z 511.566,A -85,B 0,C 180,E1 -10426.153,E2 -10426.153} C_VEL
LIN {X 0,Y 410.995,Z 515.461,A -85,B 0,C 180,E1 -10427.658,E2 -10427.658} C_VEL
LIN {X 0,Y 410.807,Z 518.267,A -85,B 0,C 180,E1 -10429.154,E2 -10429.154} C_VEL
LIN {X 0,Y 410.811,Z 519.573,A -85,B 0,C 180,E1 -10430.15,E2 -10430.15} C_VEL
LIN {X 0,Y 410.828,Z 520.412,A -85,B 0,C 180,E1 -10431.144,E2 -10431.144} C_VEL
LIN {X 0,Y 410.933,Z 520.894,A -85,B 0,C 180,E1 -10432.728,E2 -10432.728} C_VEL
LIN {X 0,Y 410.974,Z 520.432,A -85,B 0,C 180,E1 -10434.111,E2 -10434.111} C_VEL
LIN {X 0,Y 411.02,Z 519.601,A -85,B 0,C 180,E1 -10435.096,E2 -10435.096} C_VEL
LIN {X 0,Y 411.102,Z 518.361,A -85,B 0,C 180,E1 -10436.079,E2 -10436.079} C_VEL
LIN {X 0,Y 411.425,Z 515.623,A -85,B 0,C 180,E1 -10437.553,E2 -10437.553} C_VEL
LIN {X 0,Y 411.801,Z 511.828,A -85,B 0,C 180,E1 -10439.023,E2 -10439.023} C_VEL
LIN {X 0,Y 412.267,Z 506.859,A -85,B 0,C 180,E1 -10440.489,E2 -10440.489} C_VEL
LIN {X 0,Y 412.829,Z 500.575,A -85,B 0,C 180,E1 -10441.952,E2 -10441.952} C_VEL
LIN {X 0,Y 413.528,Z 492.739,A -85,B 0,C 180,E1 -10443.411,E2 -10443.411} C_VEL
LIN {X 0,Y 414.124,Z 484.677,A -85,B 0,C 180,E1 -10444.624,E2 -10444.624} C_VEL
LIN {X 0,Y 414.817,Z 474.771,A -85,B 0,C 180,E1 -10445.835,E2 -10445.835} C_VEL
LIN {X 0,Y 415.438,Z 463.766,A -85,B 0,C 180,E1 -10446.923,E2 -10446.923} C_VEL
LIN {X 0,Y 416.124,Z 451.121,A -85,B 0,C 180,E1 -10447.888,E2 -10447.888} C_VEL
LIN {X 0,Y 416.497,Z 438.583,A -85,B 0,C 180,E1 -10448.613,E2 -10448.613} C_VEL
LIN {X 0,Y 416.743,Z 425.322,A -85,B 0,C 180,E1 -10449.158,E2 -10449.158} C_VEL
LIN {X 0,Y 416.93,Z 408.267,A -85,B 0,C 180,E1 -10449.582,E2 -10449.582} C_VEL
LIN {X 0,Y 418.435,Z 346.919,A -85,B 0,C 180,E1 -10450.931,E2 -10450.931} C_VEL
LIN {X 0,Y 412.018,Z 332.627,A -85,B 0,C 180,E1 -10451.732,E2 -10451.732} C_VEL
LIN {X 0,Y 411.26,Z 330.26,A -85,B 0,C 180,E1 -10451.865,E2 -10451.865} C_VEL
LIN {X 0,Y 411.255,Z 330.258,A -85,B 0,C 180,E1 -10454.853,E2 -10454.853} C_VEL
LIN {X 0,Y 411.23,Z 330.265,A -85,B 0,C 180,E1 -10457.917,E2 -10457.917} C_VEL
LIN {X 0,Y 411.184,Z 330.269,A -85,B 0,C 180,E1 -10461.035,E2 -10461.035} C_VEL
LIN {X 0,Y 411.192,Z 330.27,A -85,B 0,C 180,E1 -10464.218,E2 -10464.218} C_VEL
LIN {X 0,Y 411.147,Z 330.271,A -85,B 0,C 180,E1 -10467.486,E2 -10467.486} C_VEL
LIN {X 0,Y 411.199,Z 330.265,A -85,B 0,C 180,E1 -10469.713,E2 -10469.713} C_VEL
LIN {X 0,Y 411.208,Z 330.261,A -85,B 0,C 180,E1 -10473.156,E2 -10473.156} C_VEL
LIN {X 0,Y 411.192,Z 330.262,A -85,B 0,C 180,E1 -10476.552,E2 -10476.552} C_VEL
LIN {X 0,Y 411.171,Z 330.265,A -85,B 0,C 180,E1 -10479.72,E2 -10479.72} C_VEL
LIN {X 0,Y 411.166,Z 330.265,A -85,B 0,C 180,E1 -10483.135,E2 -10483.135} C_VEL
LIN {X 0,Y 411.168,Z 330.269,A -85,B 0,C 180,E1 -10485.882,E2 -10485.882} C_VEL
LIN {X 0,Y 411.153,Z 330.268,A -85,B 0,C 180,E1 -10488.774,E2 -10488.774} C_VEL
LIN {X 0,Y 411.19,Z 330.267,A -85,B 0,C 180,E1 -10492.025,E2 -10492.025} C_VEL
LIN {X 0,Y 411.208,Z 330.265,A -85,B 0,C 180,E1 -10495.666,E2 -10495.666} C_VEL
LIN {X 0,Y 411.238,Z 330.394,A -85,B 0,C 180,E1 -10498.287,E2 -10498.287} C_VEL
LIN {X 0,Y 414.761,Z 346.192,A -85,B 0,C 180,E1 -10501.124,E2 -10501.124} C_VEL
LIN {X 0,Y 415.773,Z 351.369,A -85,B 0,C 180,E1 -10502.026,E2 -10502.026} C_VEL
LIN {X 0,Y 414.55,Z 369.447,A -85,B 0,C 180,E1 -10504.923,E2 -10504.923} C_VEL
LIN {X 0,Y 413.359,Z 389.082,A -85,B 0,C 180,E1 -10508.034,E2 -10508.034} C_VEL
LIN {X 0,Y 412.632,Z 403.344,A -85,B 0,C 180,E1 -10510.28,E2 -10510.28} C_VEL
LIN {X 0,Y 414.996,Z 423.791,A -85,B 0,C 180,E1 -10510.927,E2 -10510.927} C_VEL
LIN {X 0,Y 416.627,Z 441.629,A -85,B 0,C 180,E1 -10511.451,E2 -10511.451} C_VEL
LIN {X 0,Y 415.124,Z 514.643,A -85,B 0,C 180,E1 -10513.051,E2 -10513.051} C_VEL
LIN {X 0,Y 414.478,Z 528.767,A -85,B 0,C 180,E1 -10513.563,E2 -10513.563} C_VEL
LIN {X 0,Y 413.673,Z 541.405,A -85,B 0,C 180,E1 -10514.227,E2 -10514.227} C_VEL
LIN {X 0,Y 412.934,Z 553.747,A -85,B 0,C 180,E1 -10515.083,E2 -10515.083} C_VEL
LIN {X 0,Y 412.147,Z 564.877,A -85,B 0,C 180,E1 -10516.062,E2 -10516.062} C_VEL
LIN {X 0,Y 411.657,Z 575.422,A -85,B 0,C 180,E1 -10517.177,E2 -10517.177} C_VEL
LIN {X 0,Y 411.029,Z 585.181,A -85,B 0,C 180,E1 -10518.41,E2 -10518.41} C_VEL
LIN {X 0,Y 410.674,Z 593.204,A -85,B 0,C 180,E1 -10519.648,E2 -10519.648} C_VEL
LIN {X 0,Y 410.445,Z 601.021,A -85,B 0,C 180,E1 -10521.135,E2 -10521.135} C_VEL
LIN {X 0,Y 410.362,Z 607.28,A -85,B 0,C 180,E1 -10522.62,E2 -10522.62} C_VEL
LIN {X 0,Y 410.385,Z 612.192,A -85,B 0,C 180,E1 -10524.102,E2 -10524.102} C_VEL
LIN {X 0,Y 410.474,Z 615.893,A -85,B 0,C 180,E1 -10525.581,E2 -10525.581} C_VEL
LIN {X 0,Y 410.502,Z 618.473,A -85,B 0,C 180,E1 -10527.056,E2 -10527.056} C_VEL
LIN {X 0,Y 410.465,Z 619.624,A -85,B 0,C 180,E1 -10528.037,E2 -10528.037} C_VEL
LIN {X 0,Y 410.484,Z 620.292,A -85,B 0,C 180,E1 -10529.019,E2 -10529.019} C_VEL
LIN {X 0,Y 410.521,Z 620.528,A -85,B 0,C 180,E1 -10530,E2 -10530} C_VEL
LIN {X 0,Y 410.479,Z 620.324,A -85,B 0,C 180,E1 -10530.981,E2 -10530.981} C_VEL
LIN {X 0,Y 410.456,Z 619.67,A -85,B 0,C 180,E1 -10531.962,E2 -10531.962} C_VEL
LIN {X 0,Y 410.503,Z 618.557,A -85,B 0,C 180,E1 -10532.944,E2 -10532.944} C_VEL
LIN {X 0,Y 410.47,Z 616.044,A -85,B 0,C 180,E1 -10534.419,E2 -10534.419} C_VEL
LIN {X 0,Y 410.391,Z 612.453,A -85,B 0,C 180,E1 -10535.897,E2 -10535.897} C_VEL
LIN {X 0,Y 410.37,Z 607.713,A -85,B 0,C 180,E1 -10537.38,E2 -10537.38} C_VEL
LIN {X 0,Y 410.433,Z 601.698,A -85,B 0,C 180,E1 -10538.865,E2 -10538.865} C_VEL
LIN {X 0,Y 410.658,Z 594.244,A -85,B 0,C 180,E1 -10540.352,E2 -10540.352} C_VEL
LIN {X 0,Y 411.037,Z 586.703,A -85,B 0,C 180,E1 -10541.59,E2 -10541.59} C_VEL
LIN {X 0,Y 411.656,Z 577.675,A -85,B 0,C 180,E1 -10542.823,E2 -10542.823} C_VEL
LIN {X 0,Y 412.232,Z 567.828,A -85,B 0,C 180,E1 -10543.934,E2 -10543.934} C_VEL
LIN {X 0,Y 413.076,Z 555.778,A -85,B 0,C 180,E1 -10545.038,E2 -10545.038} C_VEL
LIN {X 0,Y 414.013,Z 544.045,A -85,B 0,C 180,E1 -10545.886,E2 -10545.886} C_VEL
LIN {X 0,Y 414.79,Z 530.929,A -85,B 0,C 180,E1 -10546.614,E2 -10546.614} C_VEL
LIN {X 0,Y 415.611,Z 517.504,A -85,B 0,C 180,E1 -10547.15,E2 -10547.15} C_VEL
LIN {X 0,Y 416.001,Z 500.739,A -85,B 0,C 180,E1 -10547.577,E2 -10547.577} C_VEL
LIN {X 0,Y 417.371,Z 440.225,A -85,B 0,C 180,E1 -10548.93,E2 -10548.93} C_VEL
LIN {X 0,Y 415.274,Z 416.87,A -85,B 0,C 180,E1 -10549.647,E2 -10549.647} C_VEL
LIN {X 0,Y 412.753,Z 399.17,A -85,B 0,C 180,E1 -10550.29,E2 -10550.29} C_VEL
LIN {X 0,Y 414.126,Z 378.426,A -85,B 0,C 180,E1 -10553.721,E2 -10553.721} C_VEL
LIN {X 0,Y 415.689,Z 360.003,A -85,B 0,C 180,E1 -10556.888,E2 -10556.888} C_VEL
LIN {X 0,Y 416.393,Z 352.623,A -85,B 0,C 180,E1 -10558.203,E2 -10558.203} C_VEL
LIN {X 0,Y 414.618,Z 343.178,A -85,B 0,C 180,E1 -10560.176,E2 -10560.176} C_VEL
LIN {X 0,Y 412.025,Z 333.24,A -85,B 0,C 180,E1 -10562.5,E2 -10562.5} C_VEL
LIN {X 0,Y 411.214,Z 330.266,A -85,B 0,C 180,E1 -10563.302,E2 -10563.302} C_VEL
LIN {X 0,Y 411.191,Z 330.268,A -85,B 0,C 180,E1 -10566.742,E2 -10566.742} C_VEL
LIN {X 0,Y 411.172,Z 330.27,A -85,B 0,C 180,E1 -10569.72,E2 -10569.72} C_VEL
LIN {X 0,Y 411.167,Z 330.269,A -85,B 0,C 180,E1 -10573.135,E2 -10573.135} C_VEL
LIN {X 0,Y 411.168,Z 330.27,A -85,B 0,C 180,E1 -10575.881,E2 -10575.881} C_VEL
LIN {X 0,Y 411.151,Z 330.27,A -85,B 0,C 180,E1 -10578.774,E2 -10578.774} C_VEL
LIN {X 0,Y 411.183,Z 330.266,A -85,B 0,C 180,E1 -10582.025,E2 -10582.025} C_VEL
LIN {X 0,Y 411.203,Z 330.262,A -85,B 0,C 180,E1 -10585.123,E2 -10585.123} C_VEL
LIN {X 0,Y 411.165,Z 330.27,A -85,B 0,C 180,E1 -10588.002,E2 -10588.002} C_VEL
LIN {X 0,Y 411.173,Z 330.27,A -85,B 0,C 180,E1 -10591.406,E2 -10591.406} C_VEL
LIN {X 0,Y 411.189,Z 330.267,A -85,B 0,C 180,E1 -10594.941,E2 -10594.941} C_VEL
LIN {X 0,Y 411.2,Z 330.268,A -85,B 0,C 180,E1 -10597.913,E2 -10597.913} C_VEL
LIN {X 0,Y 411.191,Z 330.268,A -85,B 0,C 180,E1 -10601.049,E2 -10601.049} C_VEL
LIN {X 0,Y 411.226,Z 330.262,A -85,B 0,C 180,E1 -10601.987,E2 -10601.987} C_VEL
LIN {X 0,Y 412.23,Z 333.14,A -85,B 0,C 180,E1 -10602.154,E2 -10602.154} C_VEL
LIN {X 0,Y 417.978,Z 345.142,A -85,B 0,C 180,E1 -10602.908,E2 -10602.908} C_VEL
LIN {X 0,Y 418.978,Z 347.778,A -85,B 0,C 180,E1 -10603.048,E2 -10603.048} C_VEL
LIN {X 0,Y 416.977,Z 419.106,A -85,B 0,C 180,E1 -10604.699,E2 -10604.699} C_VEL
LIN {X 0,Y 416.817,Z 432.939,A -85,B 0,C 180,E1 -10605.162,E2 -10605.162} C_VEL
LIN {X 0,Y 416.451,Z 446.251,A -85,B 0,C 180,E1 -10605.835,E2 -10605.835} C_VEL
LIN {X 0,Y 415.962,Z 458.776,A -85,B 0,C 180,E1 -10606.69,E2 -10606.69} C_VEL
LIN {X 0,Y 415.264,Z 469.867,A -85,B 0,C 180,E1 -10607.662,E2 -10607.662} C_VEL
LIN {X 0,Y 414.633,Z 479.882,A -85,B 0,C 180,E1 -10608.759,E2 -10608.759} C_VEL
LIN {X 0,Y 413.911,Z 489.081,A -85,B 0,C 180,E1 -10610.002,E2 -10610.002} C_VEL
LIN {X 0,Y 413.184,Z 497.652,A -85,B 0,C 180,E1 -10611.44,E2 -10611.44} C_VEL
LIN {X 0,Y 412.633,Z 504.631,A -85,B 0,C 180,E1 -10612.906,E2 -10612.906} C_VEL
LIN {X 0,Y 412.024,Z 509.341,A -85,B 0,C 180,E1 -10614.125,E2 -10614.125} C_VEL
LIN {X 0,Y 411.699,Z 513.817,A -85,B 0,C 180,E1 -10615.594,E2 -10615.594} C_VEL
LIN {X 0,Y 411.329,Z 517.192,A -85,B 0,C 180,E1 -10617.061,E2 -10617.061} C_VEL
LIN {X 0,Y 411.273,Z 518.84,A -85,B 0,C 180,E1 -10618.041,E2 -10618.041} C_VEL
LIN {X 0,Y 411.13,Z 520.048,A -85,B 0,C 180,E1 -10619.02,E2 -10619.02} C_VEL
LIN {X 0,Y 410.997,Z 520.853,A -85,B 0,C 180,E1 -10620,E2 -10620} C_VEL
LIN {X 0,Y 410.94,Z 521.243,A -85,B 0,C 180,E1 -10620.979,E2 -10620.979} C_VEL
LIN {X 0,Y 410.671,Z 521.203,A -85,B 0,C 180,E1 -10621.961,E2 -10621.961} C_VEL
LIN {X 0,Y 410.691,Z 520.724,A -85,B 0,C 180,E1 -10622.942,E2 -10622.942} C_VEL
LIN {X 0,Y 410.798,Z 519.839,A -85,B 0,C 180,E1 -10623.923,E2 -10623.923} C_VEL
LIN {X 0,Y 410.974,Z 518.502,A -85,B 0,C 180,E1 -10624.905,E2 -10624.905} C_VEL
LIN {X 0,Y 411.052,Z 515.702,A -85,B 0,C 180,E1 -10626.38,E2 -10626.38} C_VEL
LIN {X 0,Y 411.203,Z 511.838,A -85,B 0,C 180,E1 -10627.858,E2 -10627.858} C_VEL
LIN {X 0,Y 411.428,Z 506.798,A -85,B 0,C 180,E1 -10629.339,E2 -10629.339} C_VEL
LIN {X 0,Y 411.725,Z 500.43,A -85,B 0,C 180,E1 -10630.822,E2 -10630.822} C_VEL
LIN {X 0,Y 412.18,Z 492.499,A -85,B 0,C 180,E1 -10632.306,E2 -10632.306} C_VEL
LIN {X 0,Y 412.64,Z 484.35,A -85,B 0,C 180,E1 -10633.543,E2 -10633.543} C_VEL
LIN {X 0,Y 413.098,Z 474.378,A -85,B 0,C 180,E1 -10634.785,E2 -10634.785} C_VEL
LIN {X 0,Y 413.639,Z 463.303,A -85,B 0,C 180,E1 -10635.9,E2 -10635.9} C_VEL
LIN {X 0,Y 414.066,Z 452.495,A -85,B 0,C 180,E1 -10636.77,E2 -10636.77} C_VEL
LIN {X 0,Y 414.599,Z 439.611,A -85,B 0,C 180,E1 -10637.574,E2 -10637.574} C_VEL
LIN {X 0,Y 414.854,Z 426.29,A -85,B 0,C 180,E1 -10638.186,E2 -10638.186} C_VEL
LIN {X 0,Y 414.966,Z 412.756,A -85,B 0,C 180,E1 -10638.593,E2 -10638.593} C_VEL
LIN {X 0,Y 415.934,Z 344.392,A -85,B 0,C 180,E1 -10640.01,E2 -10640.01} C_VEL
LIN {X 0,Y 411.228,Z 330.263,A -85,B 0,C 180,E1 -10640.504,E2 -10640.504} C_VEL
LIN {X 0,Y 411.227,Z 330.259,A -85,B 0,C 180,E1 -10644.215,E2 -10644.215} C_VEL
LIN {X 0,Y 411.259,Z 330.255,A -85,B 0,C 180,E1 -10647.477,E2 -10647.477} C_VEL
LIN {X 0,Y 411.189,Z 330.267,A -85,B 0,C 180,E1 -10650.847,E2 -10650.847} C_VEL
LIN {X 0,Y 411.204,Z 330.263,A -85,B 0,C 180,E1 -10654.333,E2 -10654.333} C_VEL
LIN {X 0,Y 411.19,Z 330.263,A -85,B 0,C 180,E1 -10657.973,E2 -10657.973} C_VEL
LIN {X 0,Y 411.162,Z 330.267,A -85,B 0,C 180,E1 -10661.228,E2 -10661.228} C_VEL
LIN {X 0,Y 411.174,Z 330.269,A -85,B 0,C 180,E1 -10664.49,E2 -10664.49} C_VEL
LIN {X 0,Y 411.175,Z 330.266,A -85,B 0,C 180,E1 -10668.194,E2 -10668.194} C_VEL
LIN {X 0,Y 411.222,Z 330.262,A -85,B 0,C 180,E1 -10670.776,E2 -10670.776} C_VEL
LIN {X 0,Y 411.197,Z 330.267,A -85,B 0,C 180,E1 -10674.471,E2 -10674.471} C_VEL
LIN {X 0,Y 411.205,Z 330.263,A -85,B 0,C 180,E1 -10676.873,E2 -10676.873} C_VEL
LIN {X 0,Y 411.23,Z 330.262,A -85,B 0,C 180,E1 -10680.644,E2 -10680.644} C_VEL
LIN {X 0,Y 411.236,Z 330.257,A -85,B 0,C 180,E1 -10683.619,E2 -10683.619} C_VEL
LIN {X 0,Y 411.201,Z 330.263,A -85,B 0,C 180,E1 -10686.852,E2 -10686.852} C_VEL
LIN {X 0,Y 411.212,Z 330.262,A -85,B 0,C 180,E1 -10690.05,E2 -10690.05} C_VEL
LIN {X 0,Y 411.26,Z 330.255,A -85,B 0,C 180,E1 -10693.131,E2 -10693.131} C_VEL
LIN {X 0,Y 411.302,Z 330.25,A -85,B 0,C 180,E1 -10696.896,E2 -10696.896} C_VEL
LIN {X 0,Y 411.302,Z 330.253,A -85,B 0,C 180,E1 -10700.162,E2 -10700.162} C_VEL
LIN {X 0,Y 411.458,Z 330.23,A -85,B 0,C 180,E1 -10703.133,E2 -10703.133} C_VEL
LIN {X 0,Y 411.308,Z 330.249,A -85,B 0,C 180,E1 -10705.099,E2 -10705.099} C_VEL
LIN {X 0,Y 411.511,Z 330.226,A -85,B 0,C 180,E1 -10708.043,E2 -10708.043} C_VEL
LIN {X 0,Y 411.64,Z 330.21,A -85,B 0,C 180,E1 -10710,E2 -10710} C_VEL
LIN {X 0,Y 411.463,Z 330.23,A -85,B 0,C 180,E1 -10712.937,E2 -10712.937} C_VEL
LIN {X 0,Y 411.446,Z 330.233,A -85,B 0,C 180,E1 -10715.763,E2 -10715.763} C_VEL
LIN {X 0,Y 411.221,Z 330.265,A -85,B 0,C 180,E1 -10716.309,E2 -10716.309} C_VEL
LIN {X 0,Y 409.918,Z 330.432,A -85,B 0,C 180,E1 -10717.115,E2 -10717.115} C_VEL
LIN {X 0,Y 405.471,Z 330.986,A -85,B 0,C 180,E1 -10718.976,E2 -10718.976} C_VEL
LIN {X 0,Y 404.353,Z 331.12,A -85,B 0,C 180,E1 -10719.805,E2 -10719.805} C_VEL
LIN {X 0,Y 404.251,Z 331.13,A -85,B 0,C 180,E1 -10720.086,E2 -10720.086} C_VEL
LIN {X 0,Y 404.264,Z 331.126,A -85,B 0,C 180,E1 -10723.212,E2 -10723.212} C_VEL
LIN {X 0,Y 404.213,Z 331.133,A -85,B 0,C 180,E1 -10727.007,E2 -10727.007} C_VEL
LIN {X 0,Y 404.162,Z 331.141,A -85,B 0,C 180,E1 -10730.352,E2 -10730.352} C_VEL
LIN {X 0,Y 404.168,Z 331.139,A -85,B 0,C 180,E1 -10733.575,E2 -10733.575} C_VEL
LIN {X 0,Y 404.182,Z 331.139,A -85,B 0,C 180,E1 -10735.767,E2 -10735.767} C_VEL
LIN {X 0,Y 404.194,Z 331.14,A -85,B 0,C 180,E1 -10738,E2 -10738} C_VEL
LIN {X 0,Y 404.138,Z 331.143,A -85,B 0,C 180,E1 -10741.559,E2 -10741.559} C_VEL
LIN {X 0,Y 404.185,Z 331.136,A -85,B 0,C 180,E1 -10745.017,E2 -10745.017} C_VEL
LIN {X 0,Y 404.159,Z 331.14,A -85,B 0,C 180,E1 -10748.757,E2 -10748.757} C_VEL
LIN {X 0,Y 404.123,Z 331.146,A -85,B 0,C 180,E1 -10751.6,E2 -10751.6} C_VEL
LIN {X 0,Y 404.145,Z 331.142,A -85,B 0,C 180,E1 -10754.523,E2 -10754.523} C_VEL
LIN {X 0,Y 404.137,Z 331.143,A -85,B 0,C 180,E1 -10757.296,E2 -10757.296} C_VEL
LIN {X 0,Y 404.169,Z 331.141,A -85,B 0,C 180,E1 -10759.956,E2 -10759.956} C_VEL
LIN {X 0,Y 404.136,Z 331.142,A -85,B 0,C 180,E1 -10763.126,E2 -10763.126} C_VEL
LIN {X 0,Y 404.146,Z 331.143,A -85,B 0,C 180,E1 -10766.188,E2 -10766.188} C_VEL
LIN {X 0,Y 404.147,Z 331.146,A -85,B 0,C 180,E1 -10769.716,E2 -10769.716} C_VEL
LIN {X 0,Y 404.246,Z 331.131,A -85,B 0,C 180,E1 -10773.296,E2 -10773.296} C_VEL
LIN {X 0,Y 409.273,Z 346.862,A -85,B 0,C 180,E1 -10773.845,E2 -10773.845} C_VEL
LIN {X 0,Y 408.11,Z 418.607,A -85,B 0,C 180,E1 -10775.351,E2 -10775.351} C_VEL
LIN {X 0,Y 407.974,Z 430.712,A -85,B 0,C 180,E1 -10775.78,E2 -10775.78} C_VEL
LIN {X 0,Y 407.621,Z 443.937,A -85,B 0,C 180,E1 -10776.458,E2 -10776.458} C_VEL
LIN {X 0,Y 407.16,Z 456.05,A -85,B 0,C 180,E1 -10777.281,E2 -10777.281} C_VEL
LIN {X 0,Y 406.614,Z 467.833,A -85,B 0,C 180,E1 -10778.319,E2 -10778.319} C_VEL
LIN {X 0,Y 406.103,Z 477.922,A -85,B 0,C 180,E1 -10779.422,E2 -10779.422} C_VEL
LIN {X 0,Y 405.577,Z 486.206,A -85,B 0,C 180,E1 -10780.515,E2 -10780.515} C_VEL
LIN {X 0,Y 405.125,Z 494.311,A -85,B 0,C 180,E1 -10781.805,E2 -10781.805} C_VEL
LIN {X 0,Y 404.686,Z 502.146,A -85,B 0,C 180,E1 -10783.349,E2 -10783.349} C_VEL
LIN {X 0,Y 404.304,Z 508.403,A -85,B 0,C 180,E1 -10784.886,E2 -10784.886} C_VEL
LIN {X 0,Y 404.072,Z 513.294,A -85,B 0,C 180,E1 -10786.42,E2 -10786.42} C_VEL
LIN {X 0,Y 403.908,Z 516.97,A -85,B 0,C 180,E1 -10787.948,E2 -10787.948} C_VEL
LIN {X 0,Y 403.769,Z 518.807,A -85,B 0,C 180,E1 -10788.962,E2 -10788.962} C_VEL
LIN {X 0,Y 403.768,Z 520.215,A -85,B 0,C 180,E1 -10789.977,E2 -10789.977} C_VEL
LIN {X 0,Y 403.776,Z 521.171,A -85,B 0,C 180,E1 -10790.988,E2 -10790.988} C_VEL
LIN {X 0,Y 403.894,Z 521.795,A -85,B 0,C 180,E1 -10792.677,E2 -10792.677} C_VEL
LIN {X 0,Y 403.942,Z 521.479,A -85,B 0,C 180,E1 -10794.008,E2 -10794.008} C_VEL
LIN {X 0,Y 403.991,Z 520.72,A -85,B 0,C 180,E1 -10795.01,E2 -10795.01} C_VEL
LIN {X 0,Y 404.074,Z 519.564,A -85,B 0,C 180,E1 -10796.011,E2 -10796.011} C_VEL
LIN {X 0,Y 404.403,Z 516.968,A -85,B 0,C 180,E1 -10797.51,E2 -10797.51} C_VEL
LIN {X 0,Y 404.813,Z 513.326,A -85,B 0,C 180,E1 -10799.006,E2 -10799.006} C_VEL
LIN {X 0,Y 405.312,Z 508.533,A -85,B 0,C 180,E1 -10800.497,E2 -10800.497} C_VEL
LIN {X 0,Y 405.898,Z 502.409,A -85,B 0,C 180,E1 -10801.985,E2 -10801.985} C_VEL
LIN {X 0,Y 406.618,Z 494.772,A -85,B 0,C 180,E1 -10803.469,E2 -10803.469} C_VEL
LIN {X 0,Y 407.259,Z 487.006,A -85,B 0,C 180,E1 -10804.702,E2 -10804.702} C_VEL
LIN {X 0,Y 407.999,Z 477.481,A -85,B 0,C 180,E1 -10805.933,E2 -10805.933} C_VEL
LIN {X 0,Y 408.67,Z 466.871,A -85,B 0,C 180,E1 -10807.039,E2 -10807.039} C_VEL
LIN {X 0,Y 409.27,Z 456.599,A -85,B 0,C 180,E1 -10807.897,E2 -10807.897} C_VEL
LIN {X 0,Y 409.827,Z 444.324,A -85,B 0,C 180,E1 -10808.692,E2 -10808.692} C_VEL
LIN {X 0,Y 410.086,Z 431.642,A -85,B 0,C 180,E1 -10809.308,E2 -10809.308} C_VEL
LIN {X 0,Y 410.261,Z 419.343,A -85,B 0,C 180,E1 -10809.709,E2 -10809.709} C_VEL
LIN {X 0,Y 411.957,Z 348.673,A -85,B 0,C 180,E1 -10811.325,E2 -10811.325} C_VEL
LIN {X 0,Y 405.26,Z 333.967,A -85,B 0,C 180,E1 -10812.194,E2 -10812.194} C_VEL
LIN {X 0,Y 404.248,Z 331.133,A -85,B 0,C 180,E1 -10812.361,E2 -10812.361} C_VEL
LIN {X 0,Y 404.221,Z 331.135,A -85,B 0,C 180,E1 -10816.152,E2 -10816.152} C_VEL
LIN {X 0,Y 404.139,Z 331.147,A -85,B 0,C 180,E1 -10819.294,E2 -10819.294} C_VEL
LIN {X 0,Y 404.147,Z 331.141,A -85,B 0,C 180,E1 -10822.83,E2 -10822.83} C_VEL
LIN {X 0,Y 404.135,Z 331.147,A -85,B 0,C 180,E1 -10825.77,E2 -10825.77} C_VEL
LIN {X 0,Y 404.157,Z 331.141,A -85,B 0,C 180,E1 -10829.603,E2 -10829.603} C_VEL
LIN {X 0,Y 404.143,Z 331.143,A -85,B 0,C 180,E1 -10832.622,E2 -10832.622} C_VEL
LIN {X 0,Y 404.148,Z 331.137,A -85,B 0,C 180,E1 -10835.182,E2 -10835.182} C_VEL
LIN {X 0,Y 404.136,Z 331.14,A -85,B 0,C 180,E1 -10838.76,E2 -10838.76} C_VEL
LIN {X 0,Y 404.11,Z 331.144,A -85,B 0,C 180,E1 -10841.597,E2 -10841.597} C_VEL
LIN {X 0,Y 404.147,Z 331.141,A -85,B 0,C 180,E1 -10844.522,E2 -10844.522} C_VEL
LIN {X 0,Y 404.128,Z 331.145,A -85,B 0,C 180,E1 -10847.294,E2 -10847.294} C_VEL
LIN {X 0,Y 404.136,Z 331.145,A -85,B 0,C 180,E1 -10849.951,E2 -10849.951} C_VEL
LIN {X 0,Y 404.138,Z 331.144,A -85,B 0,C 180,E1 -10853.125,E2 -10853.125} C_VEL
LIN {X 0,Y 404.148,Z 331.144,A -85,B 0,C 180,E1 -10856.188,E2 -10856.188} C_VEL
LIN {X 0,Y 404.193,Z 331.237,A -85,B 0,C 180,E1 -10858.038,E2 -10858.038} C_VEL
LIN {X 0,Y 407.623,Z 346.62,A -85,B 0,C 180,E1 -10860.851,E2 -10860.851} C_VEL
LIN {X 0,Y 408.725,Z 352.013,A -85,B 0,C 180,E1 -10861.809,E2 -10861.809} C_VEL
LIN {X 0,Y 408.358,Z 360.113,A -85,B 0,C 180,E1 -10863.142,E2 -10863.142} C_VEL
LIN {X 0,Y 406.789,Z 383.031,A -85,B 0,C 180,E1 -10866.855,E2 -10866.855} C_VEL
LIN {X 0,Y 405.701,Z 401.119,A -85,B 0,C 180,E1 -10869.758,E2 -10869.758} C_VEL
LIN {X 0,Y 408.394,Z 423.512,A -85,B 0,C 180,E1 -10870.519,E2 -10870.519} C_VEL
LIN {X 0,Y 410.057,Z 442.542,A -85,B 0,C 180,E1 -10871.09,E2 -10871.09} C_VEL
LIN {X 0,Y 408.458,Z 513.592,A -85,B 0,C 180,E1 -10872.702,E2 -10872.702} C_VEL
LIN {X 0,Y 407.766,Z 527.694,A -85,B 0,C 180,E1 -10873.22,E2 -10873.22} C_VEL
LIN {X 0,Y 406.843,Z 541.332,A -85,B 0,C 180,E1 -10873.955,E2 -10873.955} C_VEL
LIN {X 0,Y 406.062,Z 553.455,A -85,B 0,C 180,E1 -10874.824,E2 -10874.824} C_VEL
LIN {X 0,Y 405.185,Z 564.392,A -85,B 0,C 180,E1 -10875.818,E2 -10875.818} C_VEL
LIN {X 0,Y 404.583,Z 574.476,A -85,B 0,C 180,E1 -10876.948,E2 -10876.948} C_VEL
LIN {X 0,Y 403.974,Z 583.733,A -85,B 0,C 180,E1 -10878.204,E2 -10878.204} C_VEL
LIN {X 0,Y 403.647,Z 591.855,A -85,B 0,C 180,E1 -10879.466,E2 -10879.466} C_VEL
LIN {X 0,Y 403.393,Z 599.787,A -85,B 0,C 180,E1 -10880.979,E2 -10880.979} C_VEL
LIN {X 0,Y 403.289,Z 606.121,A -85,B 0,C 180,E1 -10882.49,E2 -10882.49} C_VEL
LIN {X 0,Y 403.338,Z 611.104,A -85,B 0,C 180,E1 -10883.999,E2 -10883.999} C_VEL
LIN {X 0,Y 403.411,Z 614.862,A -85,B 0,C 180,E1 -10885.503,E2 -10885.503} C_VEL
LIN {X 0,Y 403.458,Z 617.494,A -85,B 0,C 180,E1 -10887.004,E2 -10887.004} C_VEL
LIN {X 0,Y 403.422,Z 618.673,A -85,B 0,C 180,E1 -10888.003,E2 -10888.003} C_VEL
LIN {X 0,Y 403.44,Z 619.376,A -85,B 0,C 180,E1 -10889.002,E2 -10889.002} C_VEL
LIN {X 0,Y 403.478,Z 619.626,A -85,B 0,C 180,E1 -10890,E2 -10890} C_VEL
LIN {X 0,Y 403.431,Z 619.437,A -85,B 0,C 180,E1 -10890.998,E2 -10890.998} C_VEL
LIN {X 0,Y 403.403,Z 618.81,A -85,B 0,C 180,E1 -10891.997,E2 -10891.997} C_VEL
LIN {X 0,Y 403.455,Z 617.711,A -85,B 0,C 180,E1 -10892.995,E2 -10892.995} C_VEL
LIN {X 0,Y 403.4,Z 615.222,A -85,B 0,C 180,E1 -10894.496,E2 -10894.496} C_VEL
LIN {X 0,Y 403.31,Z 611.651,A -85,B 0,C 180,E1 -10896.001,E2 -10896.001} C_VEL
LIN {X 0,Y 403.295,Z 606.935,A -85,B 0,C 180,E1 -10897.51,E2 -10897.51} C_VEL
LIN {X 0,Y 403.348,Z 600.954,A -85,B 0,C 180,E1 -10899.022,E2 -10899.022} C_VEL
LIN {X 0,Y 403.617,Z 593.529,A -85,B 0,C 180,E1 -10900.535,E2 -10900.535} C_VEL
LIN {X 0,Y 404.063,Z 584.384,A -85,B 0,C 180,E1 -10902.047,E2 -10902.047} C_VEL
LIN {X 0,Y 404.723,Z 574.895,A -85,B 0,C 180,E1 -10903.321,E2 -10903.321} C_VEL
LIN {X 0,Y 405.521,Z 563.675,A -85,B 0,C 180,E1 -10904.554,E2 -10904.554} C_VEL
LIN {X 0,Y 406.474,Z 552.426,A -85,B 0,C 180,E1 -10905.545,E2 -10905.545} C_VEL
LIN {X 0,Y 407.416,Z 540.041,A -85,B 0,C 180,E1 -10906.408,E2 -10906.408} C_VEL
LIN {X 0,Y 408.345,Z 527.443,A -85,B 0,C 180,E1 -10907.077,E2 -10907.077} C_VEL
LIN {X 0,Y 409.066,Z 513.804,A -85,B 0,C 180,E1 -10907.594,E2 -10907.594} C_VEL
LIN {X 0,Y 409.737,Z 489.504,A -85,B 0,C 180,E1 -10908.174,E2 -10908.174} C_VEL
LIN {X 0,Y 410.851,Z 440.379,A -85,B 0,C 180,E1 -10909.324,E2 -10909.324} C_VEL
LIN {X 0,Y 408.764,Z 417.021,A -85,B 0,C 180,E1 -10910.073,E2 -10910.073} C_VEL
LIN {X 0,Y 406.183,Z 399.793,A -85,B 0,C 180,E1 -10910.725,E2 -10910.725} C_VEL
LIN {X 0,Y 405.933,Z 397.728,A -85,B 0,C 180,E1 -10910.831,E2 -10910.831} C_VEL
LIN {X 0,Y 407.56,Z 376.461,A -85,B 0,C 180,E1 -10914.447,E2 -10914.447} C_VEL
LIN {X 0,Y 409.585,Z 355.675,A -85,B 0,C 180,E1 -10918.156,E2 -10918.156} C_VEL
LIN {X 0,Y 409.283,Z 352.118,A -85,B 0,C 180,E1 -10918.866,E2 -10918.866} C_VEL
LIN {X 0,Y 407.311,Z 342.717,A -85,B 0,C 180,E1 -10920.953,E2 -10920.953} C_VEL
LIN {X 0,Y 404.525,Z 332.605,A -85,B 0,C 180,E1 -10923.495,E2 -10923.495} C_VEL
LIN {X 0,Y 404.161,Z 331.144,A -85,B 0,C 180,E1 -10923.886,E2 -10923.886} C_VEL
LIN {X 0,Y 404.137,Z 331.146,A -85,B 0,C 180,E1 -10926.874,E2 -10926.874} C_VEL
LIN {X 0,Y 404.119,Z 331.15,A -85,B 0,C 180,E1 -10930.075,E2 -10930.075} C_VEL
LIN {X 0,Y 404.147,Z 331.144,A -85,B 0,C 180,E1 -10933.082,E2 -10933.082} C_VEL
LIN {X 0,Y 404.148,Z 331.144,A -85,B 0,C 180,E1 -10935.925,E2 -10935.925} C_VEL
LIN {X 0,Y 404.106,Z 331.149,A -85,B 0,C 180,E1 -10938.633,E2 -10938.633} C_VEL
LIN {X 0,Y 404.139,Z 331.144,A -85,B 0,C 180,E1 -10941.495,E2 -10941.495} C_VEL
LIN {X 0,Y 404.174,Z 331.138,A -85,B 0,C 180,E1 -10944.982,E2 -10944.982} C_VEL
LIN {X 0,Y 404.139,Z 331.145,A -85,B 0,C 180,E1 -10948.442,E2 -10948.442} C_VEL
LIN {X 0,Y 404.151,Z 331.142,A -85,B 0,C 180,E1 -10950.862,E2 -10950.862} C_VEL
LIN {X 0,Y 404.153,Z 331.143,A -85,B 0,C 180,E1 -10954.723,E2 -10954.723} C_VEL
LIN {X 0,Y 404.165,Z 331.145,A -85,B 0,C 180,E1 -10957.507,E2 -10957.507} C_VEL
LIN {X 0,Y 404.171,Z 331.141,A -85,B 0,C 180,E1 -10961.235,E2 -10961.235} C_VEL
LIN {X 0,Y 404.172,Z 331.14,A -85,B 0,C 180,E1 -10961.44,E2 -10961.44} C_VEL
LIN {X 0,Y 405.254,Z 334.103,A -85,B 0,C 180,E1 -10961.621,E2 -10961.621} C_VEL
LIN {X 0,Y 411.175,Z 346.184,A -85,B 0,C 180,E1 -10962.439,E2 -10962.439} C_VEL
LIN {X 0,Y 412.552,Z 349.826,A -85,B 0,C 180,E1 -10962.643,E2 -10962.643} C_VEL
LIN {X 0,Y 410.462,Z 419.872,A -85,B 0,C 180,E1 -10964.323,E2 -10964.323} C_VEL
LIN {X 0,Y 410.29,Z 433.681,A -85,B 0,C 180,E1 -10964.793,E2 -10964.793} C_VEL
LIN {X 0,Y 409.94,Z 445.986,A -85,B 0,C 180,E1 -10965.415,E2 -10965.415} C_VEL
LIN {X 0,Y 409.413,Z 457.98,A -85,B 0,C 180,E1 -10966.22,E2 -10966.22} C_VEL
LIN {X 0,Y 408.709,Z 469.464,A -85,B 0,C 180,E1 -10967.209,E2 -10967.209} C_VEL
LIN {X 0,Y 407.931,Z 480.722,A -85,B 0,C 180,E1 -10968.446,E2 -10968.446} C_VEL
LIN {X 0,Y 407.21,Z 489.64,A -85,B 0,C 180,E1 -10969.66,E2 -10969.66} C_VEL
LIN {X 0,Y 406.432,Z 497.886,A -85,B 0,C 180,E1 -10971.046,E2 -10971.046} C_VEL
LIN {X 0,Y 405.812,Z 504.99,A -85,B 0,C 180,E1 -10972.536,E2 -10972.536} C_VEL
LIN {X 0,Y 405.114,Z 510.68,A -85,B 0,C 180,E1 -10974.025,E2 -10974.025} C_VEL
LIN {X 0,Y 404.752,Z 515.071,A -85,B 0,C 180,E1 -10975.518,E2 -10975.518} C_VEL
LIN {X 0,Y 404.349,Z 518.36,A -85,B 0,C 180,E1 -10977.011,E2 -10977.011} C_VEL
LIN {X 0,Y 404.266,Z 519.934,A -85,B 0,C 180,E1 -10978.007,E2 -10978.007} C_VEL
LIN {X 0,Y 404.121,Z 521.096,A -85,B 0,C 180,E1 -10979.003,E2 -10979.003} C_VEL
LIN {X 0,Y 403.992,Z 521.859,A -85,B 0,C 180,E1 -10980,E2 -10980} C_VEL
LIN {X 0,Y 403.906,Z 522.18,A -85,B 0,C 180,E1 -10980.997,E2 -10980.997} C_VEL
LIN {X 0,Y 403.629,Z 522.091,A -85,B 0,C 180,E1 -10981.995,E2 -10981.995} C_VEL
LIN {X 0,Y 403.648,Z 521.564,A -85,B 0,C 180,E1 -10982.994,E2 -10982.994} C_VEL
LIN {X 0,Y 403.767,Z 520.619,A -85,B 0,C 180,E1 -10983.992,E2 -10983.992} C_VEL
LIN {X 0,Y 403.939,Z 519.207,A -85,B 0,C 180,E1 -10984.99,E2 -10984.99} C_VEL
LIN {X 0,Y 404.009,Z 516.311,A -85,B 0,C 180,E1 -10986.492,E2 -10986.492} C_VEL
LIN {X 0,Y 404.163,Z 512.341,A -85,B 0,C 180,E1 -10987.996,E2 -10987.996} C_VEL
LIN {X 0,Y 404.473,Z 506.22,A -85,B 0,C 180,E1 -10989.753,E2 -10989.753} C_VEL
LIN {X 0,Y 404.842,Z 499.461,A -85,B 0,C 180,E1 -10991.262,E2 -10991.262} C_VEL
LIN {X 0,Y 405.325,Z 491.006,A -85,B 0,C 180,E1 -10992.772,E2 -10992.772} C_VEL
LIN {X 0,Y 405.759,Z 482.027,A -85,B 0,C 180,E1 -10994.08,E2 -10994.08} C_VEL
LIN {X 0,Y 406.26,Z 471.708,A -85,B 0,C 180,E1 -10995.296,E2 -10995.296} C_VEL
LIN {X 0,Y 406.776,Z 461.141,A -85,B 0,C 180,E1 -10996.305,E2 -10996.305} C_VEL
LIN {X 0,Y 407.29,Z 449.63,A -85,B 0,C 180,E1 -10997.187,E2 -10997.187} C_VEL
LIN {X 0,Y 407.71,Z 436.636,A -85,B 0,C 180,E1 -10997.946,E2 -10997.946} C_VEL
LIN {X 0,Y 407.933,Z 423.025,A -85,B 0,C 180,E1 -10998.519,E2 -10998.519} C_VEL
LIN {X 0,Y 408.08,Z 408.505,A -85,B 0,C 180,E1 -10998.897,E2 -10998.897} C_VEL
LIN {X 0,Y 409.146,Z 346.057,A -85,B 0,C 180,E1 -11000.218,E2 -11000.218} C_VEL
LIN {X 0,Y 404.19,Z 331.14,A -85,B 0,C 180,E1 -11000.746,E2 -11000.746} C_VEL
LIN {X 0,Y 404.17,Z 331.138,A -85,B 0,C 180,E1 -11003.574,E2 -11003.574} C_VEL
LIN {X 0,Y 404.184,Z 331.136,A -85,B 0,C 180,E1 -11005.766,E2 -11005.766} C_VEL
LIN {X 0,Y 404.195,Z 331.134,A -85,B 0,C 180,E1 -11007.999,E2 -11007.999} C_VEL
LIN {X 0,Y 404.138,Z 331.142,A -85,B 0,C 180,E1 -11011.557,E2 -11011.557} C_VEL
LIN {X 0,Y 404.183,Z 331.138,A -85,B 0,C 180,E1 -11015.016,E2 -11015.016} C_VEL
LIN {X 0,Y 404.149,Z 331.145,A -85,B 0,C 180,E1 -11018.757,E2 -11018.757} C_VEL
LIN {X 0,Y 404.121,Z 331.144,A -85,B 0,C 180,E1 -11021.599,E2 -11021.599} C_VEL
LIN {X 0,Y 404.143,Z 331.145,A -85,B 0,C 180,E1 -11024.522,E2 -11024.522} C_VEL
LIN {X 0,Y 404.134,Z 331.142,A -85,B 0,C 180,E1 -11027.295,E2 -11027.295} C_VEL
LIN {X 0,Y 404.167,Z 331.138,A -85,B 0,C 180,E1 -11029.955,E2 -11029.955} C_VEL
LIN {X 0,Y 404.138,Z 331.142,A -85,B 0,C 180,E1 -11033.124,E2 -11033.124} C_VEL
LIN {X 0,Y 404.143,Z 331.143,A -85,B 0,C 180,E1 -11036.187,E2 -11036.187} C_VEL
LIN {X 0,Y 404.143,Z 331.141,A -85,B 0,C 180,E1 -11039.715,E2 -11039.715} C_VEL
LIN {X 0,Y 404.193,Z 331.135,A -85,B 0,C 180,E1 -11043.123,E2 -11043.123} C_VEL
LIN {X 0,Y 404.175,Z 331.137,A -85,B 0,C 180,E1 -11045.334,E2 -11045.334} C_VEL
LIN {X 0,Y 404.157,Z 331.143,A -85,B 0,C 180,E1 -11048.582,E2 -11048.582} C_VEL
LIN {X 0,Y 404.207,Z 331.133,A -85,B 0,C 180,E1 -11051.762,E2 -11051.762} C_VEL
LIN {X 0,Y 404.204,Z 331.135,A -85,B 0,C 180,E1 -11054.882,E2 -11054.882} C_VEL
LIN {X 0,Y 404.254,Z 331.129,A -85,B 0,C 180,E1 -11057.959,E2 -11057.959} C_VEL
LIN {X 0,Y 404.43,Z 331.108,A -85,B 0,C 180,E1 -11062.1,E2 -11062.1} C_VEL
LIN {X 0,Y 404.421,Z 331.109,A -85,B 0,C 180,E1 -11064.015,E2 -11064.015} C_VEL
LIN {X 0,Y 404.48,Z 331.102,A -85,B 0,C 180,E1 -11068.009,E2 -11068.009} C_VEL
LIN {X 0,Y 404.609,Z 331.086,A -85,B 0,C 180,E1 -11070,E2 -11070} C_VEL
LIN {X 0,Y 404.42,Z 331.107,A -85,B 0,C 180,E1 -11072.989,E2 -11072.989} C_VEL
LIN {X 0,Y 404.409,Z 331.109,A -85,B 0,C 180,E1 -11076.987,E2 -11076.987} C_VEL
LIN {X 0,Y 404.251,Z 331.13,A -85,B 0,C 180,E1 -11080.086,E2 -11080.086} C_VEL
LIN {X 0,Y 403.561,Z 331.214,A -85,B 0,C 180,E1 -11080.917,E2 -11080.917} C_VEL
LIN {X 0,Y 400.708,Z 331.573,A -85,B 0,C 180,E1 -11082.269,E2 -11082.269} C_VEL
LIN {X 0,Y 398.302,Z 331.875,A -85,B 0,C 180,E1 -11083.36,E2 -11083.36} C_VEL
LIN {X 0,Y 397.258,Z 332.003,A -85,B 0,C 180,E1 -11084.204,E2 -11084.204} C_VEL
LIN {X 0,Y 397.166,Z 332.012,A -85,B 0,C 180,E1 -11084.49,E2 -11084.49} C_VEL
LIN {X 0,Y 397.172,Z 332.01,A -85,B 0,C 180,E1 -11087.507,E2 -11087.507} C_VEL
LIN {X 0,Y 397.101,Z 332.019,A -85,B 0,C 180,E1 -11090.73,E2 -11090.73} C_VEL
LIN {X 0,Y 397.131,Z 332.019,A -85,B 0,C 180,E1 -11094.019,E2 -11094.019} C_VEL
LIN {X 0,Y 397.193,Z 332.007,A -85,B 0,C 180,E1 -11097.391,E2 -11097.391} C_VEL
LIN {X 0,Y 397.077,Z 332.022,A -85,B 0,C 180,E1 -11100.883,E2 -11100.883} C_VEL
LIN {X 0,Y 397.125,Z 332.017,A -85,B 0,C 180,E1 -11104.494,E2 -11104.494} C_VEL
LIN {X 0,Y 397.106,Z 332.02,A -85,B 0,C 180,E1 -11108.275,E2 -11108.275} C_VEL
LIN {X 0,Y 397.089,Z 332.02,A -85,B 0,C 180,E1 -11110.909,E2 -11110.909} C_VEL
LIN {X 0,Y 397.101,Z 332.021,A -85,B 0,C 180,E1 -11113.649,E2 -11113.649} C_VEL
LIN {X 0,Y 397.102,Z 332.019,A -85,B 0,C 180,E1 -11116.522,E2 -11116.522} C_VEL
LIN {X 0,Y 397.113,Z 332.018,A -85,B 0,C 180,E1 -11120.423,E2 -11120.423} C_VEL
LIN {X 0,Y 397.108,Z 332.019,A -85,B 0,C 180,E1 -11124.266,E2 -11124.266} C_VEL
LIN {X 0,Y 397.115,Z 332.017,A -85,B 0,C 180,E1 -11126.728,E2 -11126.728} C_VEL
LIN {X 0,Y 397.126,Z 332.017,A -85,B 0,C 180,E1 -11130.297,E2 -11130.297} C_VEL
LIN {X 0,Y 397.212,Z 332.018,A -85,B 0,C 180,E1 -11133.05,E2 -11133.05} C_VEL
LIN {X 0,Y 402.348,Z 347.442,A -85,B 0,C 180,E1 -11133.594,E2 -11133.594} C_VEL
LIN {X 0,Y 401.16,Z 419.97,A -85,B 0,C 180,E1 -11135.162,E2 -11135.162} C_VEL
LIN {X 0,Y 401.038,Z 432.135,A -85,B 0,C 180,E1 -11135.614,E2 -11135.614} C_VEL
LIN {X 0,Y 400.641,Z 445.839,A -85,B 0,C 180,E1 -11136.343,E2 -11136.343} C_VEL
LIN {X 0,Y 400.202,Z 457.131,A -85,B 0,C 180,E1 -11137.137,E2 -11137.137} C_VEL
LIN {X 0,Y 399.632,Z 468.856,A -85,B 0,C 180,E1 -11138.192,E2 -11138.192} C_VEL
LIN {X 0,Y 399.084,Z 479.453,A -85,B 0,C 180,E1 -11139.378,E2 -11139.378} C_VEL
LIN {X 0,Y 398.432,Z 488.905,A -85,B 0,C 180,E1 -11140.687,E2 -11140.687} C_VEL
LIN {X 0,Y 397.927,Z 498.095,A -85,B 0,C 180,E1 -11142.263,E2 -11142.263} C_VEL
LIN {X 0,Y 397.503,Z 505.339,A -85,B 0,C 180,E1 -11143.832,E2 -11143.832} C_VEL
LIN {X 0,Y 397.116,Z 511.951,A -85,B 0,C 180,E1 -11145.655,E2 -11145.655} C_VEL
LIN {X 0,Y 396.943,Z 516.338,A -85,B 0,C 180,E1 -11147.276,E2 -11147.276} C_VEL
LIN {X 0,Y 396.734,Z 519.326,A -85,B 0,C 180,E1 -11148.764,E2 -11148.764} C_VEL
LIN {X 0,Y 396.71,Z 520.815,A -85,B 0,C 180,E1 -11149.796,E2 -11149.796} C_VEL
LIN {X 0,Y 396.741,Z 521.897,A -85,B 0,C 180,E1 -11150.827,E2 -11150.827} C_VEL
LIN {X 0,Y 396.854,Z 522.699,A -85,B 0,C 180,E1 -11152.626,E2 -11152.626} C_VEL
LIN {X 0,Y 396.914,Z 522.49,A -85,B 0,C 180,E1 -11153.902,E2 -11153.902} C_VEL
LIN {X 0,Y 396.963,Z 521.84,A -85,B 0,C 180,E1 -11154.922,E2 -11154.922} C_VEL
LIN {X 0,Y 397.045,Z 520.753,A -85,B 0,C 180,E1 -11155.94,E2 -11155.94} C_VEL
LIN {X 0,Y 397.278,Z 519.239,A -85,B 0,C 180,E1 -11156.958,E2 -11156.958} C_VEL
LIN {X 0,Y 397.681,Z 516.097,A -85,B 0,C 180,E1 -11158.481,E2 -11158.481} C_VEL
LIN {X 0,Y 398.16,Z 511.873,A -85,B 0,C 180,E1 -11160,E2 -11160} C_VEL
LIN {X 0,Y 398.877,Z 505.356,A -85,B 0,C 180,E1 -11161.767,E2 -11161.767} C_VEL
LIN {X 0,Y 399.533,Z 498.283,A -85,B 0,C 180,E1 -11163.278,E2 -11163.278} C_VEL
LIN {X 0,Y 400.259,Z 491.001,A -85,B 0,C 180,E1 -11164.532,E2 -11164.532} C_VEL
LIN {X 0,Y 400.971,Z 482.147,A -85,B 0,C 180,E1 -11165.785,E2 -11165.785} C_VEL
LIN {X 0,Y 401.831,Z 471.186,A -85,B 0,C 180,E1 -11167.033,E2 -11167.033} C_VEL
LIN {X 0,Y 402.515,Z 460.104,A -85,B 0,C 180,E1 -11168.03,E2 -11168.03} C_VEL
LIN {X 0,Y 403.176,Z 447.762,A -85,B 0,C 180,E1 -11168.9,E2 -11168.9} C_VEL
LIN {X 0,Y 403.514,Z 435.341,A -85,B 0,C 180,E1 -11169.556,E2 -11169.556} C_VEL
LIN {X 0,Y 403.75,Z 422.514,A -85,B 0,C 180,E1 -11170.025,E2 -11170.025} C_VEL
LIN {X 0,Y 405.021,Z 371.699,A -85,B 0,C 180,E1 -11171.213,E2 -11171.213} C_VEL
LIN {X 0,Y 405.554,Z 350.525,A -85,B 0,C 180,E1 -11171.727,E2 -11171.727} C_VEL
LIN {X 0,Y 398.414,Z 335.102,A -85,B 0,C 180,E1 -11172.704,E2 -11172.704} C_VEL
LIN {X 0,Y 397.292,Z 332.298,A -85,B 0,C 180,E1 -11172.876,E2 -11172.876} C_VEL
LIN {X 0,Y 397.239,Z 332.006,A -85,B 0,C 180,E1 -11172.956,E2 -11172.956} C_VEL
LIN {X 0,Y 397.168,Z 332.013,A -85,B 0,C 180,E1 -11176.447,E2 -11176.447} C_VEL
LIN {X 0,Y 397.116,Z 332.021,A -85,B 0,C 180,E1 -11180.285,E2 -11180.285} C_VEL
LIN {X 0,Y 397.109,Z 332.022,A -85,B 0,C 180,E1 -11184.02,E2 -11184.02} C_VEL
LIN {X 0,Y 397.067,Z 332.025,A -85,B 0,C 180,E1 -11187.4,E2 -11187.4} C_VEL
LIN {X 0,Y 397.102,Z 332.022,A -85,B 0,C 180,E1 -11189.863,E2 -11189.863} C_VEL
LIN {X 0,Y 397.116,Z 332.017,A -85,B 0,C 180,E1 -11193.273,E2 -11193.273} C_VEL
LIN {X 0,Y 397.097,Z 332.016,A -85,B 0,C 180,E1 -11196.996,E2 -11196.996} C_VEL
LIN {X 0,Y 397.058,Z 332.022,A -85,B 0,C 180,E1 -11200.437,E2 -11200.437} C_VEL
LIN {X 0,Y 397.091,Z 332.022,A -85,B 0,C 180,E1 -11203.651,E2 -11203.651} C_VEL
LIN {X 0,Y 397.102,Z 332.02,A -85,B 0,C 180,E1 -11206.522,E2 -11206.522} C_VEL
LIN {X 0,Y 397.09,Z 332.022,A -85,B 0,C 180,E1 -11210.419,E2 -11210.419} C_VEL
LIN {X 0,Y 397.1,Z 332.02,A -85,B 0,C 180,E1 -11213.005,E2 -11213.005} C_VEL
LIN {X 0,Y 397.122,Z 332.019,A -85,B 0,C 180,E1 -11216.282,E2 -11216.282} C_VEL
LIN {X 0,Y 397.144,Z 332.069,A -85,B 0,C 180,E1 -11217.784,E2 -11217.784} C_VEL
LIN {X 0,Y 400.721,Z 348.184,A -85,B 0,C 180,E1 -11220.78,E2 -11220.78} C_VEL
LIN {X 0,Y 401.828,Z 353.961,A -85,B 0,C 180,E1 -11221.82,E2 -11221.82} C_VEL
LIN {X 0,Y 400.773,Z 368.745,A -85,B 0,C 180,E1 -11224.277,E2 -11224.277} C_VEL
LIN {X 0,Y 399.35,Z 389.987,A -85,B 0,C 180,E1 -11227.767,E2 -11227.767} C_VEL
LIN {X 0,Y 398.844,Z 398.953,A -85,B 0,C 180,E1 -11229.232,E2 -11229.232} C_VEL
LIN {X 0,Y 401.794,Z 422.945,A -85,B 0,C 180,E1 -11230.074,E2 -11230.074} C_VEL
LIN {X 0,Y 403.519,Z 443.347,A -85,B 0,C 180,E1 -11230.716,E2 -11230.716} C_VEL
LIN {X 0,Y 401.796,Z 512.963,A -85,B 0,C 180,E1 -11232.34,E2 -11232.34} C_VEL
